// Конвейер шнековый 30330
	dks_shnek_30330:= x4_30;
	dp_shnek_30330:= NOT x4_31;
	localstop_shnek_30330:= NOT x5_0;
	erraz_shnek_30330:= NOT x5_1;
	localpusk_shnek_30330:= x5_2;
	y7_8:= run_shnek_30330;
	
// Затвор шлюзовый 30340
	dks_shluz_30340:= x5_3;
	erraz_shluz_30340:= NOT x5_4;
	y7_9:= run_shluz_30340;
	
// Конвейер скребковый 30400
	dks_sktr_30400:= x5_5;
	dp_sktr_30400:= NOT x5_6;
	localpusk_sktr_30400:= x5_7;
	localstop_sktr_30400:= NOT x5_8;
	localstop_end_sktr_30400:= NOT x5_9;
	erraz_sktr_30400:= NOT x5_10;
	y7_10:= run_sktr_30400;
	
// Нория 30500
	dks_noria_30500:= x5_11;
	dsl1_noria_30500:= NOT x5_12;
	dsl2_noria_30500:= NOT x5_13;
	dp_noria_30500:= NOT x5_14;
	localpusk_noria_30500:= x5_15;
	localstop_but_noria_30500:= NOT x5_16;
	localstop_top_noria_30500:= NOT x5_17;
	erraz_noria_30500:= NOT x5_18;
	y7_11:= run_noria_30500;	
	
// Датчики уровня бункеров смесителя
	TON_28(IN:= NOT x5_19, PT:= WORD_TO_TIME(timeDVY_load*100), Q=> dvy_bunk_30610);
	TON_29(IN:= NOT x5_20, PT:= WORD_TO_TIME(timeDNU_load*100), Q=> dny_bunk_30610);
	TON_30(IN:= NOT x5_21, PT:= WORD_TO_TIME(timeDNU_load*100), Q=> dny_bunk_30630);
	
// Датчик открытия люка на бункере БО-5	
	open_door_bunk_BO5:= x3_31;
	
// Смеситель горизонтальный СГП-1000 (30600)
	open_door_smes:= NOT x5_22;
	dks_smes:= x5_23;
	erraz_smes:= NOT x5_24;
	y7_12:= run_smes;
	
// от смесителя поворотный клапана, бомба люк
	klap_revers_open:= NOT x5_25;
	klap_revers_close:= NOT x5_26;
	shtok_1_left_open:= NOT x5_27;
	shtok_1_left_close:= NOT x5_28;
	shtok_2_left_open:= NOT x5_29;
	shtok_2_left_close:= NOT x5_30;
	shtok_1_right_open:= NOT x5_31;
	shtok_1_right_close:= NOT a2x0_0;
	shtok_2_right_open:= NOT a2x0_1;
	shtok_2_right_close:= NOT a2x0_2;
	shtok_1_zamok_close:= NOT a2x0_3;
	shtok_1_zamok_open:= NOT a2x0_4;
	shtok_2_zamok_close:= NOT a2x0_5;
	shtok_2_zamok_open:= NOT a2x0_6;
	signal_err_smes:= NOT a2x0_7;
	
	y7_13:= run_klap_revers_open;
	y7_14:= run_shtok_left_open;
	y7_15:= run_shtok_left_close;
	y7_16:= run_shtok_right_open;
	y7_17:= run_shtok_right_close;
	y7_18:= run_open_zamok;
	y7_19:= run_close_zamok;
	
// Конвейер шнековый 30640
	dks_shnek_30640:= a2x0_8;
	dp_shnek_30640:= NOT a2x0_9;
	localstop_shnek30640:= NOT a2x0_10;
	erraz_shnek_30640:= NOT a2x0_11;
	localpusk_shnek_30640:= a2x0_12;
	y7_20:= run_shnek_30640;
	
// Вентиляция аспирации АС7
	erraz_AC_7:= NOT a2x0_13;
	y7_21:= run_AC_7;
	
// Затвор шлюзовой аспирации АС-7_1
	dks_shluz_AC_7_1:= a2x0_14;
	erraz_shluz_AC_7_1:= NOT a2x0_15;
	y7_22:= run_shluz_AC_7_1;
	
// Затвор шлюзовой аспирации АС-7_2
	dks_shluz_AC_7_2:= a2x0_16;
	erraz_shluz_AC_7_2:= NOT a2x0_17;
	y7_23:= run_shluz_AC_7_2;
	
// Нория 30700
	dks_noria_30700:= a2x0_18;
	dsl1_noria_30700:= NOT a2x0_19;
	dsl2_noria_30700:= NOT a2x0_20;
	dp_noria_30700:= NOT a2x0_21;
	localpusk_noria_30700:= a2x0_22;
	localstop_but_noria_30700:= NOT a2x0_23;
	localstop_top_noria_30700:= NOT a2x3_0;
	erraz_noria_30700:= NOT a2x3_1;
	y7_24:= run_noria_30700;
	
// Система аспирации АС-8 (30701)
	erraz_AC_30701:= NOT a2x3_2;
	y7_25:= run_AC_30701;
	
// Конвейер скребковый 30900
	dp_sktr_30900:= NOT a2x3_3;
	localpusk_sktr_30900:= a2x3_4;
	localstop_sktr_30900:= NOT a2x3_5;
	erraz_sktr_30900:= NOT a2x3_6;
	dks_sktr_30900:= NOT a2x3_7;
	localstop_end_sktr_30900:= NOT a2x3_8;
	y7_26:= run_sktr_30900;
	
// Система аспирации АС-9 (30901)
	erraz_AC_30901:= NOT a2x3_9;
	y7_27:= run_AC_30901;
	
// Шибер конвейера 30900 (30910)
	opened_sh_30910:= NOT a2x3_10;
	closed_sh_30910:= NOT a2x3_11;
	erraz_sh_30910:= NOT a2x3_12;
	y7_28:= run_open_sh_30910;
	y7_29:= run_close_sh_30910;
	
// Шибер конвейера 30900 (30920)
	opened_sh_30920:= NOT a2x3_13;
	closed_sh_30920:= NOT a2x3_14;
	erraz_sh_30920:= NOT a2x3_15;
	y7_30:= run_open_sh_30920;
	y7_31:= run_close_sh_30920;
	
// Шибер конвейера 30900 (30930)
	opened_sh_30930:= NOT a2x3_16;
	closed_sh_30930:= NOT a2x3_17;
	erraz_sh_30930:= NOT a2x3_18;
	a2y0_0:= run_open_sh_30930;
	a2y0_1:= run_close_sh_30930;
	
// Шибер конвейера 30900 (30940)
	opened_sh_30940:= NOT a2x3_19;
	closed_sh_30940:= NOT a2x3_20;
	erraz_sh_30940:= NOT a2x3_21;
	a2y0_2:= run_open_sh_30940;
	a2y0_3:= run_close_sh_30940;
	
// Конвейер скребковыйй 30800
	dks_sktr_30800:= a2x3_22;
	dp_sktr_30800:= NOT a2x3_23;
	localpusk_sktr_30800:= a2x3_24;
	localstop_sktr_30800:= NOT a2x3_25;
	localstop_end_sktr_30800:= NOT a2x3_26;
	erraz_sktr_30800:= NOT a2x3_27;
	a2y0_4:= run_sktr_30800;
	
// Шибер конвейера 30800 (30810)
	opened_sh_30810:= NOT a2x3_28;
	closed_sh_30810:= NOT a2x3_29;
	erraz_sh_30810:= NOT a2x3_30;
	a2y0_5:= run_open_sh_30810;
	a2y0_6:= run_close_sh_30810;
	
// Конвейер бункера малых весов
	dks_shnek_21600:= a2x3_31;
	dp_shnek_21600:= NOT a2x4_0;
	localstop_21600:= NOT a2x4_1;
	erraz_shnek_21600:= NOT a2x4_2;
	localpusk_shnek_21600:= a2x4_3;
	a2y0_7:= run_shnek_21600;
	
// скальператор барабанный 10300
	errpch_scalp:= a2x4_4;
	a2y0_8:= run_scalp;
	a2y0_9:= run_resset_pch_scalp;
	a2y0_10:= run_pch_scalp;
	
// Дазаторы 20011-20016
	errpch_doz_11_16:= a2x4_5;
	a2y0_11:= run_pch_doz_11_16;
	a2y0_12:= run_resset_pch_doz_11_16;
	
	a2y0_13:= run_doz_shnek_20011;
	a2y0_14:= run_doz_shnek_20012;
	a2y0_15:= run_doz_shnek_20013;
	a2y6_0:= run_doz_shnek_20014;
	a2y6_1:= run_doz_shnek_20015;
	a2y6_2:= run_doz_shnek_20016;
	
	dp_doz_shnek_20011:= NOT a2x4_6;
	localstop_doz_shnek_20011:= NOT a2x4_7;
	dp_doz_shnek_20012:= NOT a2x4_8;
	localstop_doz_shnek_20012:= NOT a2x4_9;
	dp_doz_shnek_20013:= NOT a2x4_10;
	localstop_doz_shnek_20013:= NOT a2x4_11;
	dp_doz_shnek_20014:= NOT a2x4_12;
	localstop_doz_shnek_20014:= NOT a2x4_13;
	dp_doz_shnek_20015:= NOT a2x4_14;
	localstop_doz_shnek_20015:= NOT a2x4_15;
	dp_doz_shnek_20016:= NOT a2x4_16;
	localstop_doz_shnek_20016:= NOT a2x4_17;
	
// Дазаторы 20017-20018
	errpch_doz_17_18:= a2x4_18;
	a2y6_3:= run_pch_doz_17_18;
	a2y6_4:= run_resset_pch_doz_17_18;
	
	a2y6_5:= run_doz_shnek_20017;
	a2y6_6:= run_doz_shnek_20018;
	
	dp_doz_shnek_20017:= NOT a2x4_19;
	localstop_doz_shnek_20017:= NOT a2x4_20;
	dp_doz_shnek_20018:= NOT a2x4_21;
	localstop_doz_shnek_20018:= NOT a2x4_22;
	
// Дазатор 21510-21540
	errpch_doz_shnek_51_54:= a2x4_23;
	a2y6_7:= run_pch_doz_shnek_51_54;
	a2y6_8:= run_resset_pch_doz_shnek_51_54;
	
	a2y6_9:= run_doz_shnek_21510;
	a2y6_10:= run_doz_shnek_21520;
	a2y6_11:= run_doz_shnek_21530;
	a2y6_12:= run_doz_shnek_21540;
	
	dp_doz_shnek_21510:= NOT a2x4_24;
	localstop_doz_shnek_21510:= NOT a2x4_25;
	dp_doz_shnek_21520:= NOT a2x4_26;
	localstop_doz_shnek_21520:= NOT a2x4_27;
	dp_doz_shnek_21530:= NOT a2x4_28;
	localstop_doz_shnek_21530:= NOT a2x4_29;
	dp_doz_shnek_21540:= NOT a2x4_30;
	localstop_doz_shnek_21540:= NOT a2x4_31;
	
// Дазатор 21405-21409
	errpch_doz_shnek_5_9:= a2x5_0;
	a2y6_13:= run_pch_doz_shnek_5_9;
	a2y6_14:= run_resset_pch_doz_shnek_5_9;
	
	a2y6_15:= run_doz_shnek_21405;
	a2y6_16:= run_doz_shnek_21406;
	a2y6_17:= run_doz_shnek_21407;
	a2y6_18:= run_doz_shnek_21408;
	a2y6_19:= run_doz_shnek_21409;
	
	localstop_doz_shnek_21405:= NOT a2x5_1;
	localstop_doz_shnek_21406:= NOT a2x5_2;
	localstop_doz_shnek_21407:= NOT a2x5_3;
	localstop_doz_shnek_21408:= NOT a2x5_4;
	localstop_doz_shnek_21409:= NOT a2x5_5;
	
// Датчики верхнего уровня готовой продукции
	TON_31(IN:= NOT a2x5_6, PT:= WORD_TO_TIME(timeDVY_load*100), Q=> dvy_bunk_401);
	TON_32(IN:= NOT a2x5_7, PT:= WORD_TO_TIME(timeDVY_load*100), Q=> dvy_bunk_402);
	TON_33(IN:= NOT a2x5_8, PT:= WORD_TO_TIME(timeDVY_load*100), Q=> dvy_bunk_403);
	TON_34(IN:= NOT a2x5_9, PT:= WORD_TO_TIME(timeDVY_load*100), Q=> dvy_bunk_404);
	TON_35(IN:= NOT a2x5_10, PT:= WORD_TO_TIME(timeDVY_load*100), Q=> dvy_bunk_405);
	TON_36(IN:= NOT a2x5_11, PT:= WORD_TO_TIME(timeDVY_load*100), Q=> dvy_bunk_406);

// Датчики нижнего уровня готовой продукции
	TON_37(IN:= NOT a2x5_12, PT:= WORD_TO_TIME(timeDNU_load*100), Q=> dny_bunk_401);
	TON_38(IN:= NOT a2x5_13, PT:= WORD_TO_TIME(timeDNU_load*100), Q=> dny_bunk_402);
	TON_39(IN:= NOT a2x5_14, PT:= WORD_TO_TIME(timeDNU_load*100), Q=> dny_bunk_403);
	TON_40(IN:= NOT a2x5_15, PT:= WORD_TO_TIME(timeDNU_load*100), Q=> dny_bunk_404);
	TON_41(IN:= NOT a2x5_16, PT:= WORD_TO_TIME(timeDNU_load*100), Q=> dny_bunk_405);
	TON_42(IN:= NOT a2x5_17, PT:= WORD_TO_TIME(timeDNU_load*100), Q=> dny_bunk_406);
	
// Вентиляторы фильтр-шкафоф завальной ямы
	localpusk_fan_hole:= a2x5_18;
	localstop_fan_hole:= NOT a2x5_19;
	erraz_AC1_1_1:= NOT a2x5_20;
	erraz_AC2_1_1:= NOT a2x5_21;
	erraz_AC3_1_1:= NOT a2x5_22;
	erraz_AC1_1_2:= NOT a2x5_23;
	erraz_AC2_1_2:= NOT a2x5_24;
	erraz_AC3_1_2:= NOT a2x5_25;
	a2y6_20:= run_fans_AC_hole;
	
// Датчик нижнего уровня завальной ямы
	TON_43(IN:= NOT a2x5_26, PT:= WORD_TO_TIME(timeDNU_load*100), Q=> dny_hole);
	
// Конвейер 30330
	errpch_sktr_30330:= a2x5_27;
	a2y6_21:= run_pch_sktr_30330;
	a2y6_22:= run_resset_pch_sktr_30330;
	
// Конвейер 30640
	errpch_sktr_30640:= a2x5_28;
	a2y6_23:= run_pch_sktr_30640;
	a2y6_24:= run_resset_pch_sktr_30640;
	
// Весы большие
	W1_Big:= %IW39;
	W2_Big:= %IW40;
	Weight_Big.WordValue[0]:= W2_Big;
	Weight_Big.WordValue[1]:= W1_Big;
	CurrWeight_Big:= Weight_Big.RealValue-Tare_big_weight;
	
// Весы средние
	W1_Midle:= %IW41;
	W2_Midle:= %IW42;
	Weight_Midle.WordValue[0]:= W2_Midle;
	Weight_Midle.WordValue[1]:= W1_Midle;
	CurrWeight_Midle:= Weight_Midle.RealValue-Tare_midle_weight;

END_PROGRAM

// PLC_241/Application/POU/prgLoad
PROGRAM prgLoad
VAR
	T_SKTR_10110: T;
	AC_10201: AC;
	N_10200: N;
	KP_10210: KP;
	SCLP_10300: SCLP;
	AC_10401: AC;
	N_10400: N;
	AC_10501: AC;
	T_10500: T;
	Z_10610: Z;
	KP_10710: KP;
	Z_10620: Z;
	KP_10720: KP;
	Z_10630: Z;
	KP_10730: KP;
	Z_10640: Z;
	KP_10740: KP;
	AC_fans_hole: AC;
	TP_STEP: TP;
	Step: WORD;
	imp: BOOL;
	imp_dvy_101: BOOL;
	imp_dvy_102: BOOL;
	imp_dvy_103: BOOL;
	imp_dvy_104: BOOL;
	imp_dvy_105: BOOL;
	imp_dvy_106: BOOL;
	imp_dvy_107: BOOL;
	imp_dvy_108: BOOL;
	pause_load: BOOL;
	TON_pause: TON;
	TOF_next_sktr_10500: TOF;
	TON_imp_bunk_101: TON;
	TON_imp_bunk_102: TON;
	timePause_load_queu3: TON;
	TON_imp_bunk_103: TON;
	TON_imp_bunk_104: TON;
	TON_imp_bunk_105: TON;
	TON_imp_bunk_107: TON;
	TON_imp_bunk_106: TON;
	TON_imp_bunk_108: TON;
	TON_pause_DNY_HOLE: TON;
	use_time_hole: BOOL;
	TON_RESSET_modeLoad: TON;
	check: BOOL;
	TON_nextBunk: TON;
	imp_nextBunk: BOOL;
END_VAR
VAR // added by the converter: edge detectors and wires of the graphical bodies
    _rt1, _rt2, _rt3, _rt4, _rt5, _rt6, _rt7, _rt8, _rt9, _rt10, _rt11, _rt12, _rt13, _rt14, _rt15, _rt16, _rt17, _rt18, _rt19, _rt20, _rt21 : R_TRIG;
    _w1, _w2, _w3, _w4, _w5, _w6, _w7, _w8, _w9, _w10 : BOOL;
END_VAR

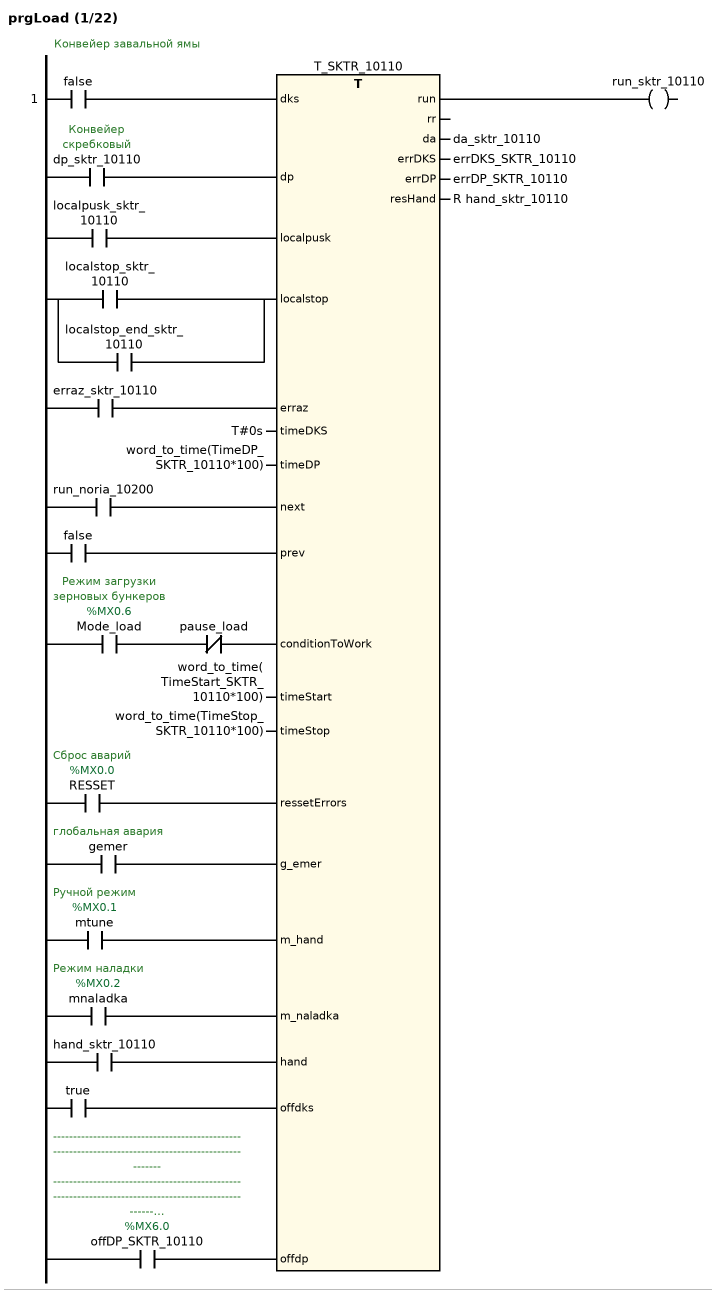
// NETWORK 1
// Конвейер завальной ямы
//   dp_sktr_10110: Конвейер скребковый
//   Mode_load: Режим загрузки зерновых бункеров | AT %MX0.6
//   RESSET: Сброс аварий | AT %MX0.0
//   gemer: глобальная авария
//   mtune: Ручной режим | AT %MX0.1
//   mnaladka: Режим наладки | AT %MX0.2
//   offDP_SKTR_10110: ----------------------------------------------------------------------------------------------------- ----------------------------------------------------------------------------------------------------- Отключение датчиков из скады ----------------------------------------------------------------------------------------------------- Конвейер завальной ямы | AT %MX6.0
//   errDKS_SKTR_10110: Конвейер завальной ямы 10110
T_SKTR_10110(
    dks := false,
    dp := dp_sktr_10110,
    localpusk := localpusk_sktr_10110,
    localstop := localstop_sktr_10110 OR localstop_end_sktr_10110,
    erraz := erraz_sktr_10110,
    timeDKS := T#0s,
    timeDP := word_to_time(TimeDP_SKTR_10110*100),
    next := run_noria_10200,
    prev := false,
    conditionToWork := Mode_load AND NOT pause_load,
    timeStart := word_to_time(TimeStart_SKTR_10110*100),
    timeStop := word_to_time(TimeStop_SKTR_10110*100),
    ressetErrors := RESSET,
    g_emer := gemer,
    m_hand := mtune,
    m_naladka := mnaladka,
    hand := hand_sktr_10110,
    offdks := true,
    offdp := offDP_SKTR_10110,
    da => da_sktr_10110,
    errDKS => errDKS_SKTR_10110,
    errDP => errDP_SKTR_10110); // T
hand_sktr_10110 R= T_SKTR_10110.resHand;
run_sktr_10110 := T_SKTR_10110.run;

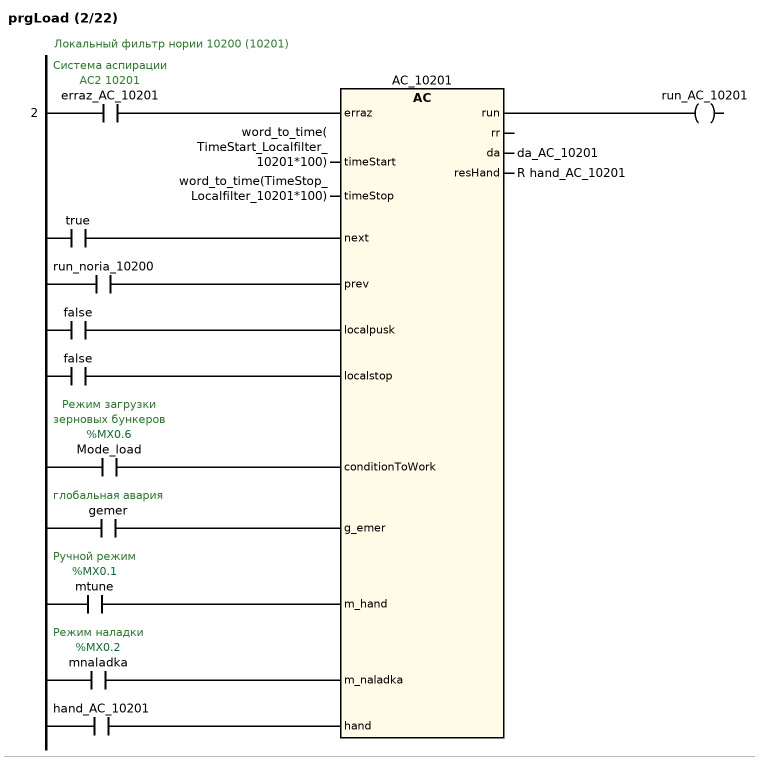
// NETWORK 2
// Локальный фильтр нории 10200 (10201)
//   erraz_AC_10201: Система аспирации АС2 10201
//   Mode_load: Режим загрузки зерновых бункеров | AT %MX0.6
//   gemer: глобальная авария
//   mtune: Ручной режим | AT %MX0.1
//   mnaladka: Режим наладки | AT %MX0.2
AC_10201(
    erraz := erraz_AC_10201,
    timeStart := word_to_time(TimeStart_Localfilter_10201*100),
    timeStop := word_to_time(TimeStop_Localfilter_10201*100),
    next := true,
    prev := run_noria_10200,
    localpusk := false,
    localstop := false,
    conditionToWork := Mode_load,
    g_emer := gemer,
    m_hand := mtune,
    m_naladka := mnaladka,
    hand := hand_AC_10201,
    da => da_AC_10201); // AC
hand_AC_10201 R= AC_10201.resHand;
run_AC_10201 := AC_10201.run;

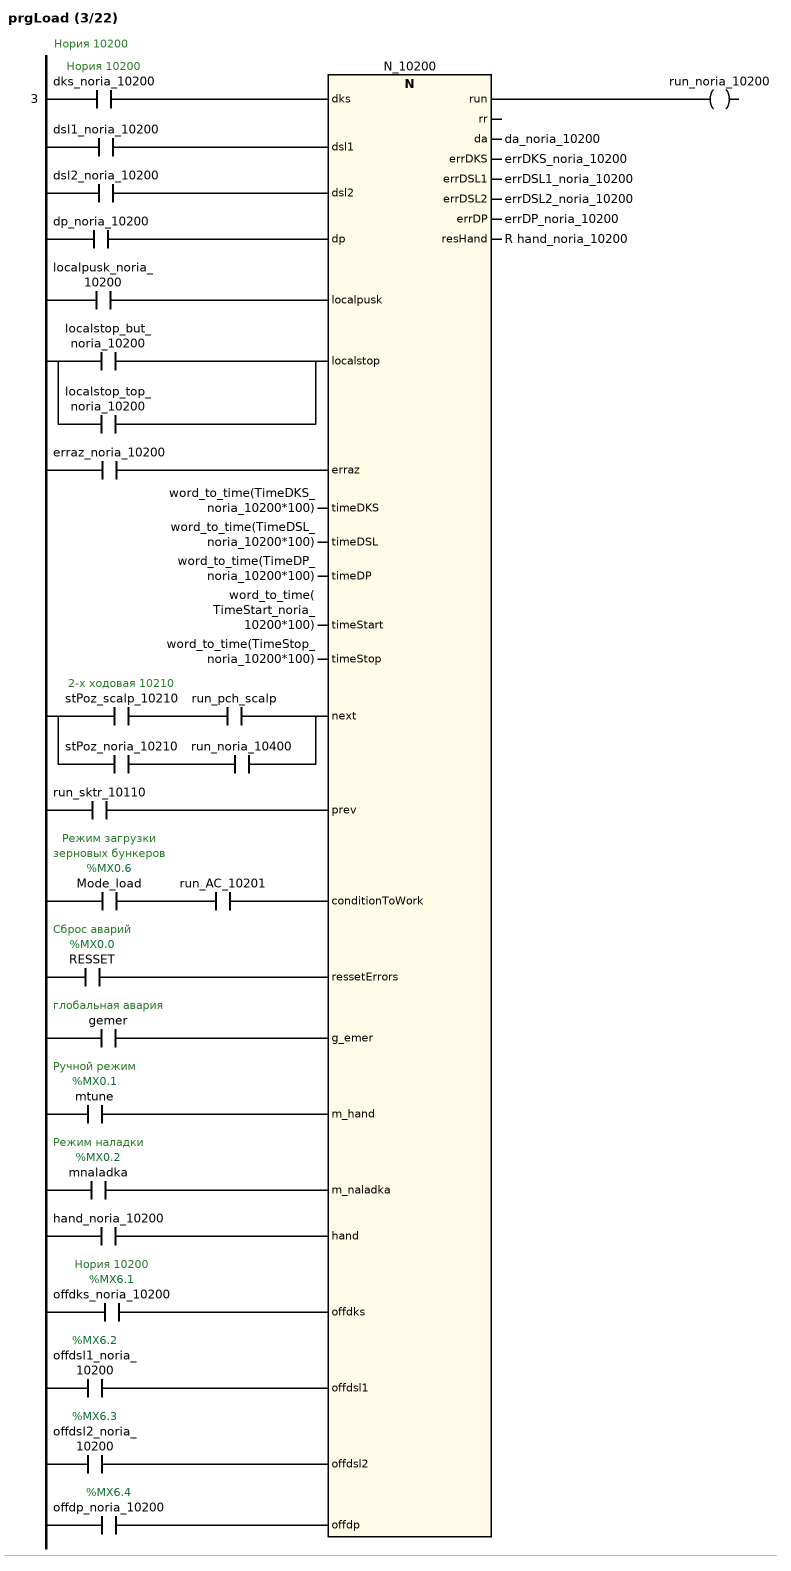
// NETWORK 3
// Нория 10200
//   dks_noria_10200: Нория 10200
//   stPoz_scalp_10210: 2-х ходовая 10210
//   Mode_load: Режим загрузки зерновых бункеров | AT %MX0.6
//   RESSET: Сброс аварий | AT %MX0.0
//   gemer: глобальная авария
//   mtune: Ручной режим | AT %MX0.1
//   mnaladka: Режим наладки | AT %MX0.2
//   offdks_noria_10200: Нория 10200 | AT %MX6.1
//   offdsl1_noria_10200: AT %MX6.2
//   offdsl2_noria_10200: AT %MX6.3
//   offdp_noria_10200: AT %MX6.4
//   errDKS_noria_10200: Нория 10200
N_10200(
    dks := dks_noria_10200,
    dsl1 := dsl1_noria_10200,
    dsl2 := dsl2_noria_10200,
    dp := dp_noria_10200,
    localpusk := localpusk_noria_10200,
    localstop := localstop_but_noria_10200 OR localstop_top_noria_10200,
    erraz := erraz_noria_10200,
    timeDKS := word_to_time(TimeDKS_noria_10200*100),
    timeDSL := word_to_time(TimeDSL_noria_10200*100),
    timeDP := word_to_time(TimeDP_noria_10200*100),
    timeStart := word_to_time(TimeStart_noria_10200*100),
    timeStop := word_to_time(TimeStop_noria_10200*100),
    next := stPoz_scalp_10210 AND run_pch_scalp OR stPoz_noria_10210 AND run_noria_10400,
    prev := run_sktr_10110,
    conditionToWork := Mode_load AND run_AC_10201,
    ressetErrors := RESSET,
    g_emer := gemer,
    m_hand := mtune,
    m_naladka := mnaladka,
    hand := hand_noria_10200,
    offdks := offdks_noria_10200,
    offdsl1 := offdsl1_noria_10200,
    offdsl2 := offdsl2_noria_10200,
    offdp := offdp_noria_10200,
    da => da_noria_10200,
    errDKS => errDKS_noria_10200,
    errDSL1 => errDSL1_noria_10200,
    errDSL2 => errDSL2_noria_10200,
    errDP => errDP_noria_10200); // N
hand_noria_10200 R= N_10200.resHand;
run_noria_10200 := N_10200.run;

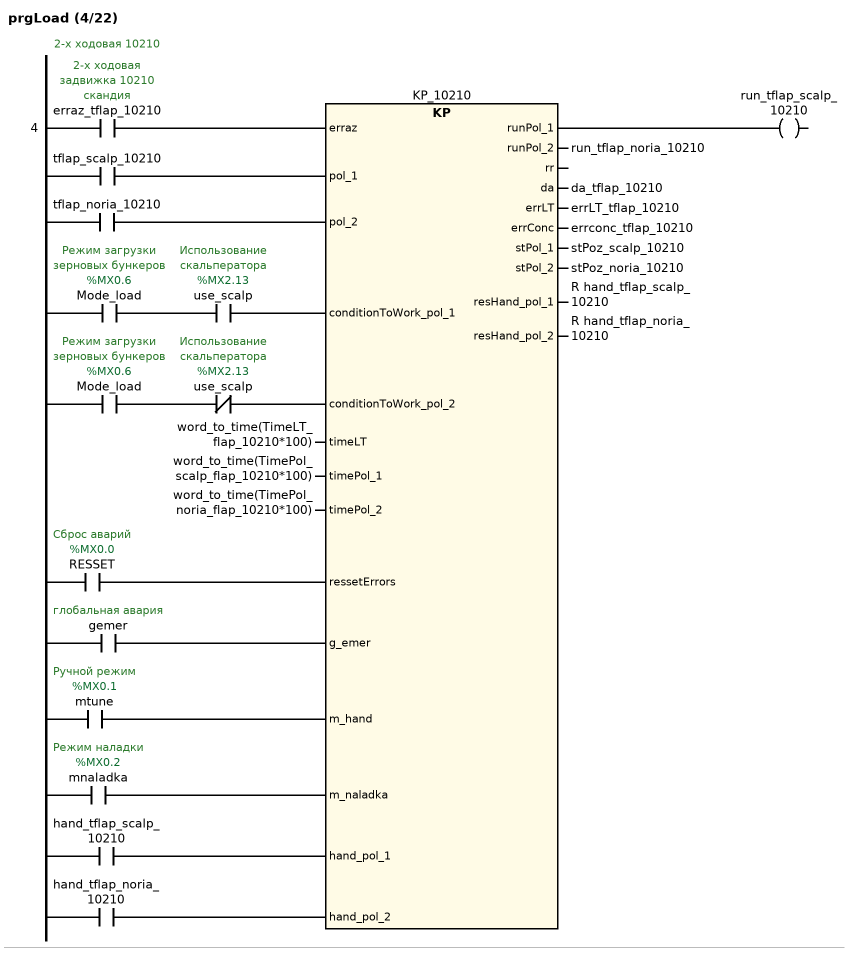
// NETWORK 4
// 2-х ходовая 10210
//   erraz_tflap_10210: 2-х ходовая задвижка 10210 скандия
//   Mode_load: Режим загрузки зерновых бункеров | AT %MX0.6
//   use_scalp: Использование скальператора | AT %MX2.13
//   RESSET: Сброс аварий | AT %MX0.0
//   gemer: глобальная авария
//   mtune: Ручной режим | AT %MX0.1
//   mnaladka: Режим наладки | AT %MX0.2
//   errLT_tflap_10210: 2-х ходовой клапан КП_10210
//   stPoz_scalp_10210: 2-х ходовая 10210
KP_10210(
    erraz := erraz_tflap_10210,
    pol_1 := tflap_scalp_10210,
    pol_2 := tflap_noria_10210,
    conditionToWork_pol_1 := Mode_load AND use_scalp,
    conditionToWork_pol_2 := Mode_load AND NOT use_scalp,
    timeLT := word_to_time(TimeLT_flap_10210*100),
    timePol_1 := word_to_time(TimePol_scalp_flap_10210*100),
    timePol_2 := word_to_time(TimePol_noria_flap_10210*100),
    ressetErrors := RESSET,
    g_emer := gemer,
    m_hand := mtune,
    m_naladka := mnaladka,
    hand_pol_1 := hand_tflap_scalp_10210,
    hand_pol_2 := hand_tflap_noria_10210,
    runPol_2 => run_tflap_noria_10210,
    da => da_tflap_10210,
    errLT => errLT_tflap_10210,
    errConc => errconc_tflap_10210,
    stPol_1 => stPoz_scalp_10210,
    stPol_2 => stPoz_noria_10210); // KP
hand_tflap_scalp_10210 R= KP_10210.resHand_pol_1;
hand_tflap_noria_10210 R= KP_10210.resHand_pol_2;
run_tflap_scalp_10210 := KP_10210.runPol_1;

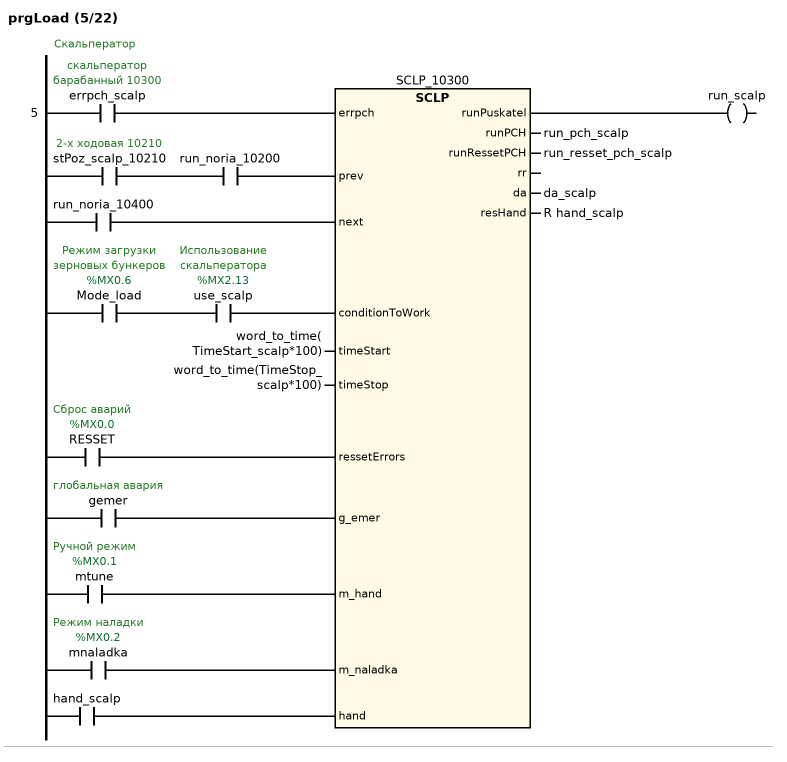
// NETWORK 5
// Скальператор
//   errpch_scalp: скальператор барабанный 10300
//   stPoz_scalp_10210: 2-х ходовая 10210
//   Mode_load: Режим загрузки зерновых бункеров | AT %MX0.6
//   use_scalp: Использование скальператора | AT %MX2.13
//   RESSET: Сброс аварий | AT %MX0.0
//   gemer: глобальная авария
//   mtune: Ручной режим | AT %MX0.1
//   mnaladka: Режим наладки | AT %MX0.2
SCLP_10300(
    errpch := errpch_scalp,
    prev := stPoz_scalp_10210 AND run_noria_10200,
    next := run_noria_10400,
    conditionToWork := Mode_load AND use_scalp,
    timeStart := word_to_time(TimeStart_scalp*100),
    timeStop := word_to_time(TimeStop_scalp*100),
    ressetErrors := RESSET,
    g_emer := gemer,
    m_hand := mtune,
    m_naladka := mnaladka,
    hand := hand_scalp,
    runPCH => run_pch_scalp,
    runRessetPCH => run_resset_pch_scalp,
    da => da_scalp); // SCLP
hand_scalp R= SCLP_10300.resHand;
run_scalp := SCLP_10300.runPuskatel;

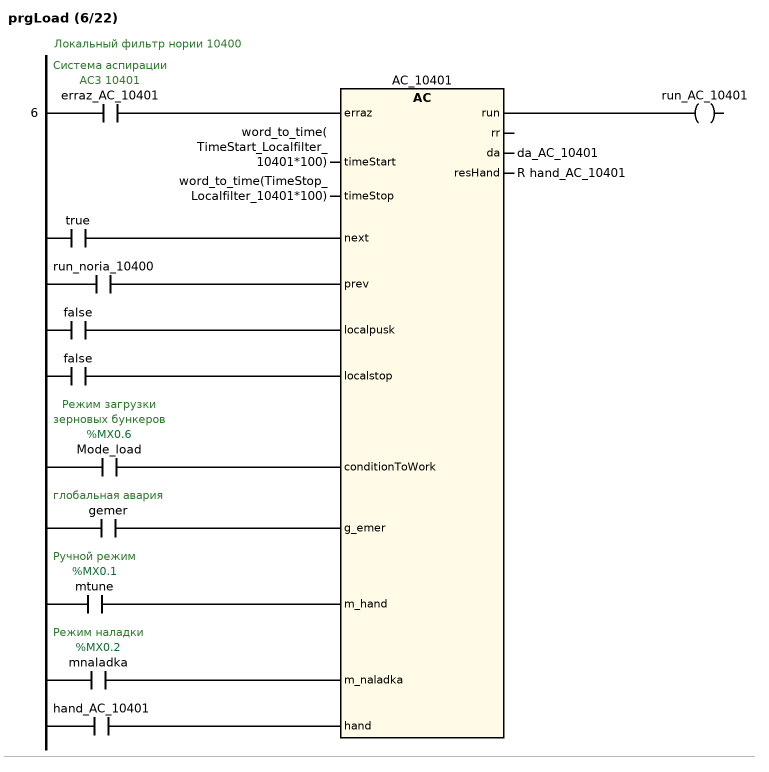
// NETWORK 6
// Локальный фильтр нории 10400
//   erraz_AC_10401: Система аспирации АС3 10401
//   Mode_load: Режим загрузки зерновых бункеров | AT %MX0.6
//   gemer: глобальная авария
//   mtune: Ручной режим | AT %MX0.1
//   mnaladka: Режим наладки | AT %MX0.2
AC_10401(
    erraz := erraz_AC_10401,
    timeStart := word_to_time(TimeStart_Localfilter_10401*100),
    timeStop := word_to_time(TimeStop_Localfilter_10401*100),
    next := true,
    prev := run_noria_10400,
    localpusk := false,
    localstop := false,
    conditionToWork := Mode_load,
    g_emer := gemer,
    m_hand := mtune,
    m_naladka := mnaladka,
    hand := hand_AC_10401,
    da => da_AC_10401); // AC
hand_AC_10401 R= AC_10401.resHand;
run_AC_10401 := AC_10401.run;

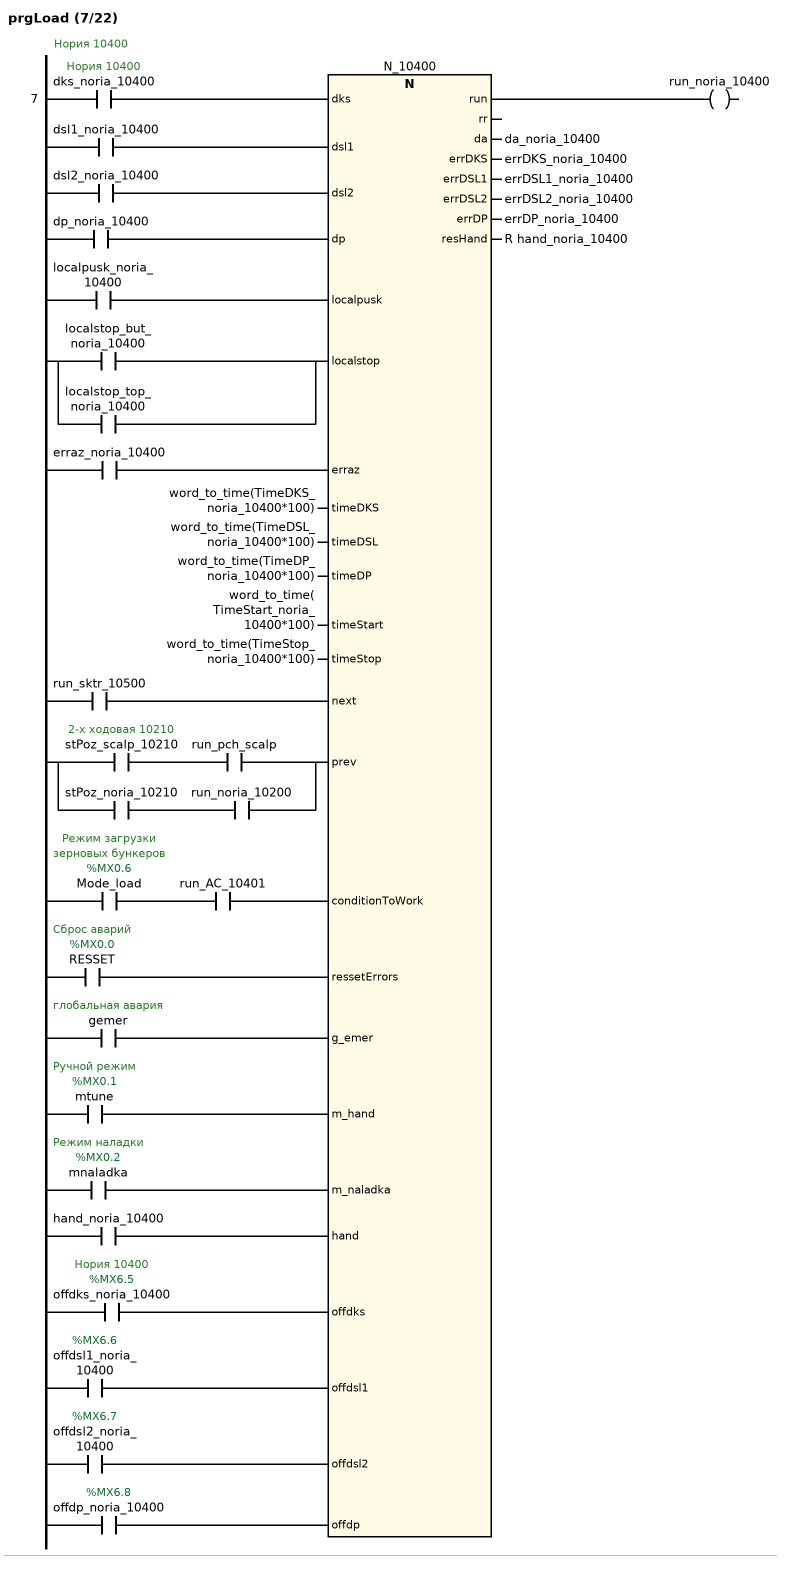
// NETWORK 7
// Нория 10400
//   dks_noria_10400: Нория 10400
//   stPoz_scalp_10210: 2-х ходовая 10210
//   Mode_load: Режим загрузки зерновых бункеров | AT %MX0.6
//   RESSET: Сброс аварий | AT %MX0.0
//   gemer: глобальная авария
//   mtune: Ручной режим | AT %MX0.1
//   mnaladka: Режим наладки | AT %MX0.2
//   offdks_noria_10400: Нория 10400 | AT %MX6.5
//   offdsl1_noria_10400: AT %MX6.6
//   offdsl2_noria_10400: AT %MX6.7
//   offdp_noria_10400: AT %MX6.8
//   errDKS_noria_10400: Нория 10400
N_10400(
    dks := dks_noria_10400,
    dsl1 := dsl1_noria_10400,
    dsl2 := dsl2_noria_10400,
    dp := dp_noria_10400,
    localpusk := localpusk_noria_10400,
    localstop := localstop_but_noria_10400 OR localstop_top_noria_10400,
    erraz := erraz_noria_10400,
    timeDKS := word_to_time(TimeDKS_noria_10400*100),
    timeDSL := word_to_time(TimeDSL_noria_10400*100),
    timeDP := word_to_time(TimeDP_noria_10400*100),
    timeStart := word_to_time(TimeStart_noria_10400*100),
    timeStop := word_to_time(TimeStop_noria_10400*100),
    next := run_sktr_10500,
    prev := stPoz_scalp_10210 AND run_pch_scalp OR stPoz_noria_10210 AND run_noria_10200,
    conditionToWork := Mode_load AND run_AC_10401,
    ressetErrors := RESSET,
    g_emer := gemer,
    m_hand := mtune,
    m_naladka := mnaladka,
    hand := hand_noria_10400,
    offdks := offdks_noria_10400,
    offdsl1 := offdsl1_noria_10400,
    offdsl2 := offdsl2_noria_10400,
    offdp := offdp_noria_10400,
    da => da_noria_10400,
    errDKS => errDKS_noria_10400,
    errDSL1 => errDSL1_noria_10400,
    errDSL2 => errDSL2_noria_10400,
    errDP => errDP_noria_10400); // N
hand_noria_10400 R= N_10400.resHand;
run_noria_10400 := N_10400.run;

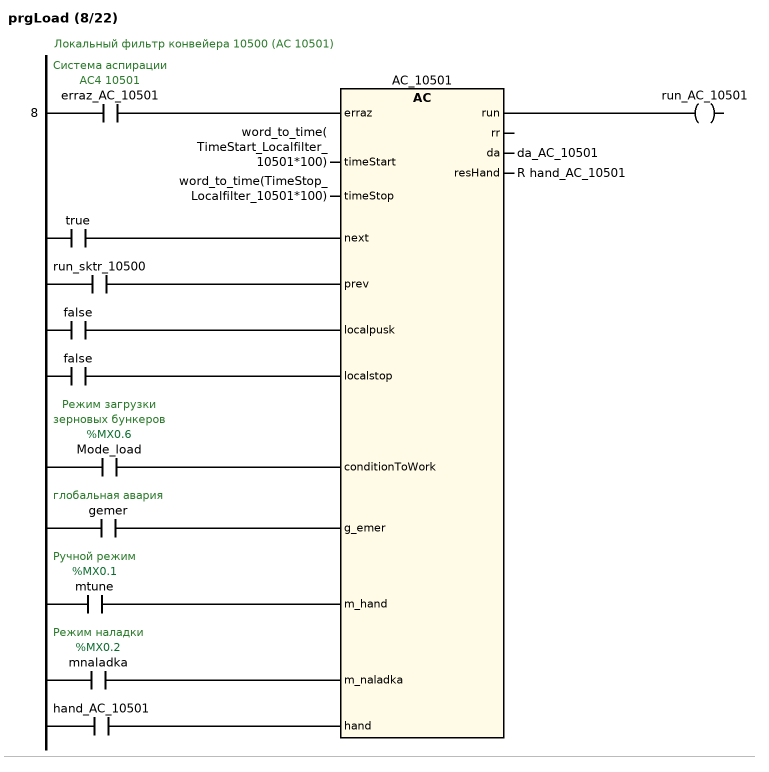
// NETWORK 8
// Локальный фильтр конвейера 10500 (АС 10501)
//   erraz_AC_10501: Система аспирации АС4 10501
//   Mode_load: Режим загрузки зерновых бункеров | AT %MX0.6
//   gemer: глобальная авария
//   mtune: Ручной режим | AT %MX0.1
//   mnaladka: Режим наладки | AT %MX0.2
AC_10501(
    erraz := erraz_AC_10501,
    timeStart := word_to_time(TimeStart_Localfilter_10501*100),
    timeStop := word_to_time(TimeStop_Localfilter_10501*100),
    next := true,
    prev := run_sktr_10500,
    localpusk := false,
    localstop := false,
    conditionToWork := Mode_load,
    g_emer := gemer,
    m_hand := mtune,
    m_naladka := mnaladka,
    hand := hand_AC_10501,
    da => da_AC_10501); // AC
hand_AC_10501 R= AC_10501.resHand;
run_AC_10501 := AC_10501.run;

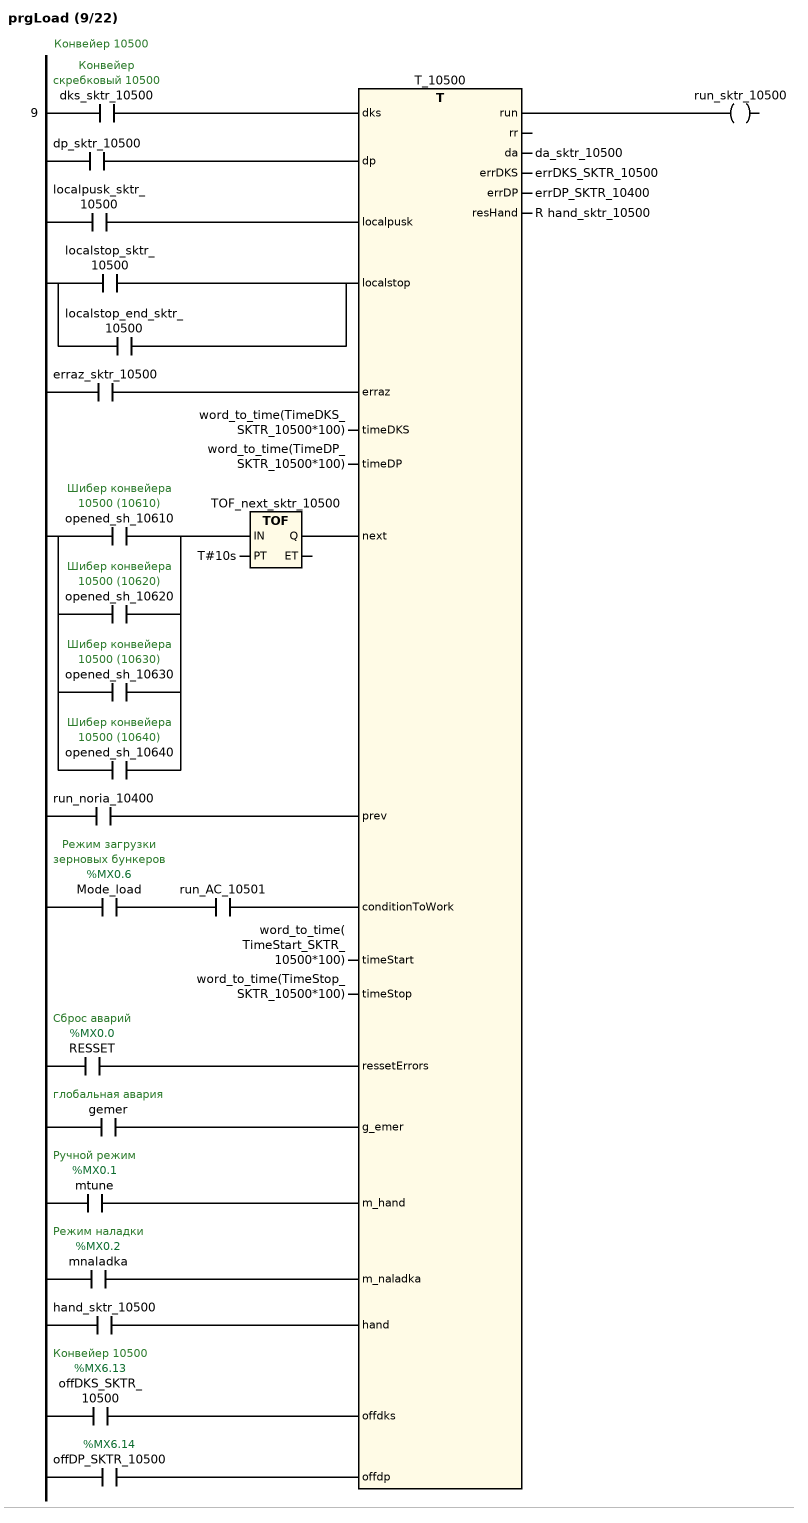
// NETWORK 9
// Конвейер 10500
//   dks_sktr_10500: Конвейер скребковый 10500
//   opened_sh_10610: Шибер конвейера 10500 (10610)
//   opened_sh_10620: Шибер конвейера 10500 (10620)
//   opened_sh_10630: Шибер конвейера 10500 (10630)
//   opened_sh_10640: Шибер конвейера 10500 (10640)
//   Mode_load: Режим загрузки зерновых бункеров | AT %MX0.6
//   RESSET: Сброс аварий | AT %MX0.0
//   gemer: глобальная авария
//   mtune: Ручной режим | AT %MX0.1
//   mnaladka: Режим наладки | AT %MX0.2
//   offDKS_SKTR_10500: Конвейер 10500 | AT %MX6.13
//   offDP_SKTR_10500: AT %MX6.14
//   errDKS_SKTR_10500: Конвейер 10500
TOF_next_sktr_10500(IN := opened_sh_10610 OR opened_sh_10620 OR opened_sh_10630 OR opened_sh_10640, PT := T#10s); // TOF
T_10500(
    dks := dks_sktr_10500,
    dp := dp_sktr_10500,
    localpusk := localpusk_sktr_10500,
    localstop := localstop_sktr_10500 OR localstop_end_sktr_10500,
    erraz := erraz_sktr_10500,
    timeDKS := word_to_time(TimeDKS_SKTR_10500*100),
    timeDP := word_to_time(TimeDP_SKTR_10500*100),
    next := TOF_next_sktr_10500.Q,
    prev := run_noria_10400,
    conditionToWork := Mode_load AND run_AC_10501,
    timeStart := word_to_time(TimeStart_SKTR_10500*100),
    timeStop := word_to_time(TimeStop_SKTR_10500*100),
    ressetErrors := RESSET,
    g_emer := gemer,
    m_hand := mtune,
    m_naladka := mnaladka,
    hand := hand_sktr_10500,
    offdks := offDKS_SKTR_10500,
    offdp := offDP_SKTR_10500,
    da => da_sktr_10500,
    errDKS => errDKS_SKTR_10500,
    errDP => errDP_SKTR_10400); // T
hand_sktr_10500 R= T_10500.resHand;
run_sktr_10500 := T_10500.run;

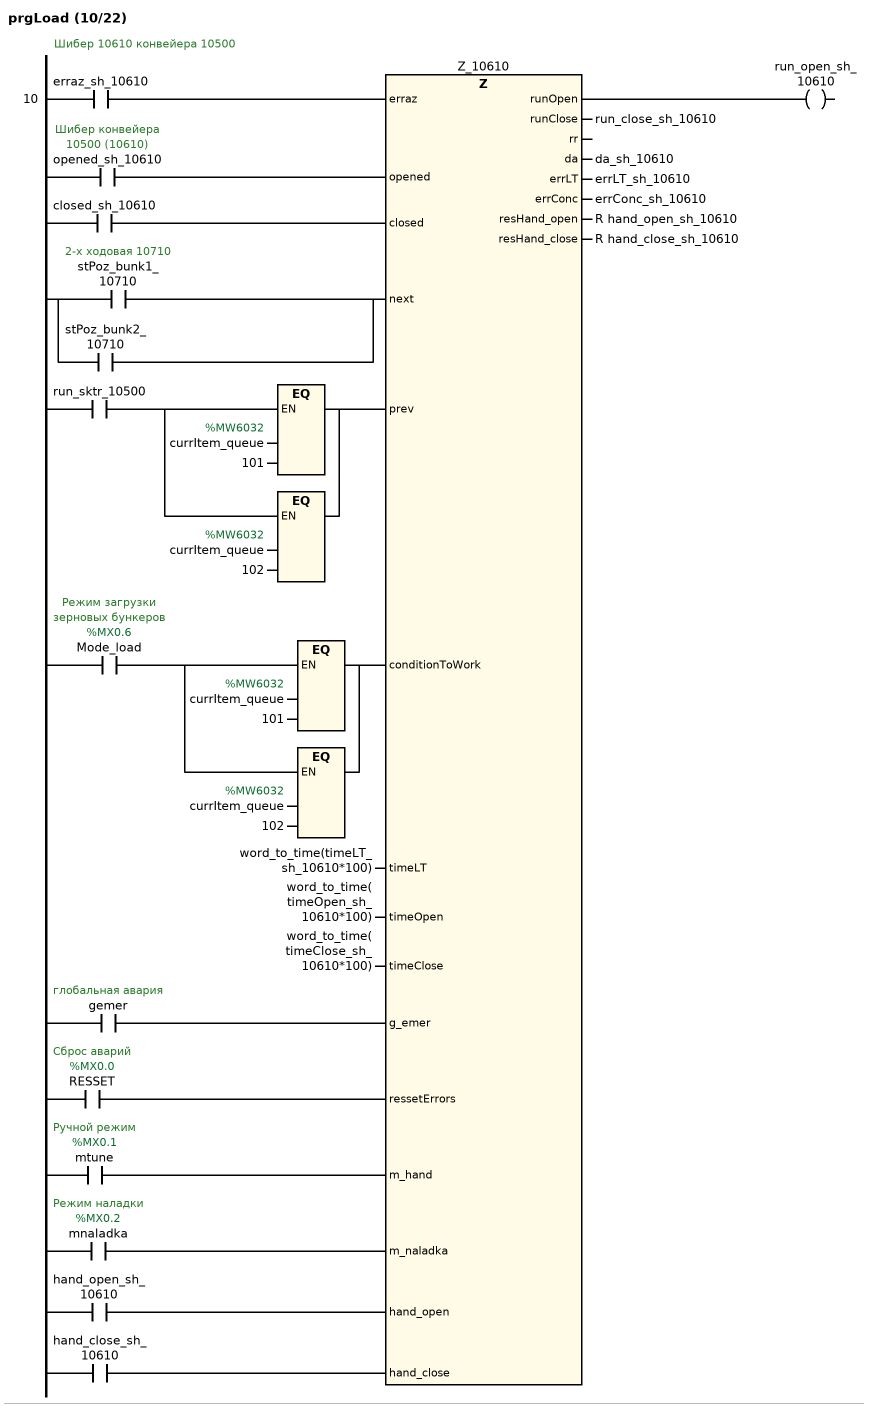
// NETWORK 10
// Шибер 10610 конвейера 10500
//   opened_sh_10610: Шибер конвейера 10500 (10610)
//   stPoz_bunk1_10710: 2-х ходовая 10710
//   currItem_queue: Текущий бункер для загрузки в очереди | AT %MW6032
//   Mode_load: Режим загрузки зерновых бункеров | AT %MX0.6
//   gemer: глобальная авария
//   RESSET: Сброс аварий | AT %MX0.0
//   mtune: Ручной режим | AT %MX0.1
//   mnaladka: Режим наладки | AT %MX0.2
//   errLT_sh_10610: Шибер 10610
Z_10610(
    erraz := erraz_sh_10610,
    opened := opened_sh_10610,
    closed := closed_sh_10610,
    next := stPoz_bunk1_10710 OR stPoz_bunk2_10710,
    prev := run_sktr_10500 AND currItem_queue = 101 OR run_sktr_10500 AND currItem_queue = 102,
    conditionToWork := Mode_load AND currItem_queue = 101 OR Mode_load AND currItem_queue = 102,
    timeLT := word_to_time(timeLT_sh_10610*100),
    timeOpen := word_to_time(timeOpen_sh_10610*100),
    timeClose := word_to_time(timeClose_sh_10610*100),
    g_emer := gemer,
    ressetErrors := RESSET,
    m_hand := mtune,
    m_naladka := mnaladka,
    hand_open := hand_open_sh_10610,
    hand_close := hand_close_sh_10610,
    runClose => run_close_sh_10610,
    da => da_sh_10610,
    errLT => errLT_sh_10610,
    errConc => errConc_sh_10610); // Z
hand_open_sh_10610 R= Z_10610.resHand_open;
hand_close_sh_10610 R= Z_10610.resHand_close;
run_open_sh_10610 := Z_10610.runOpen;

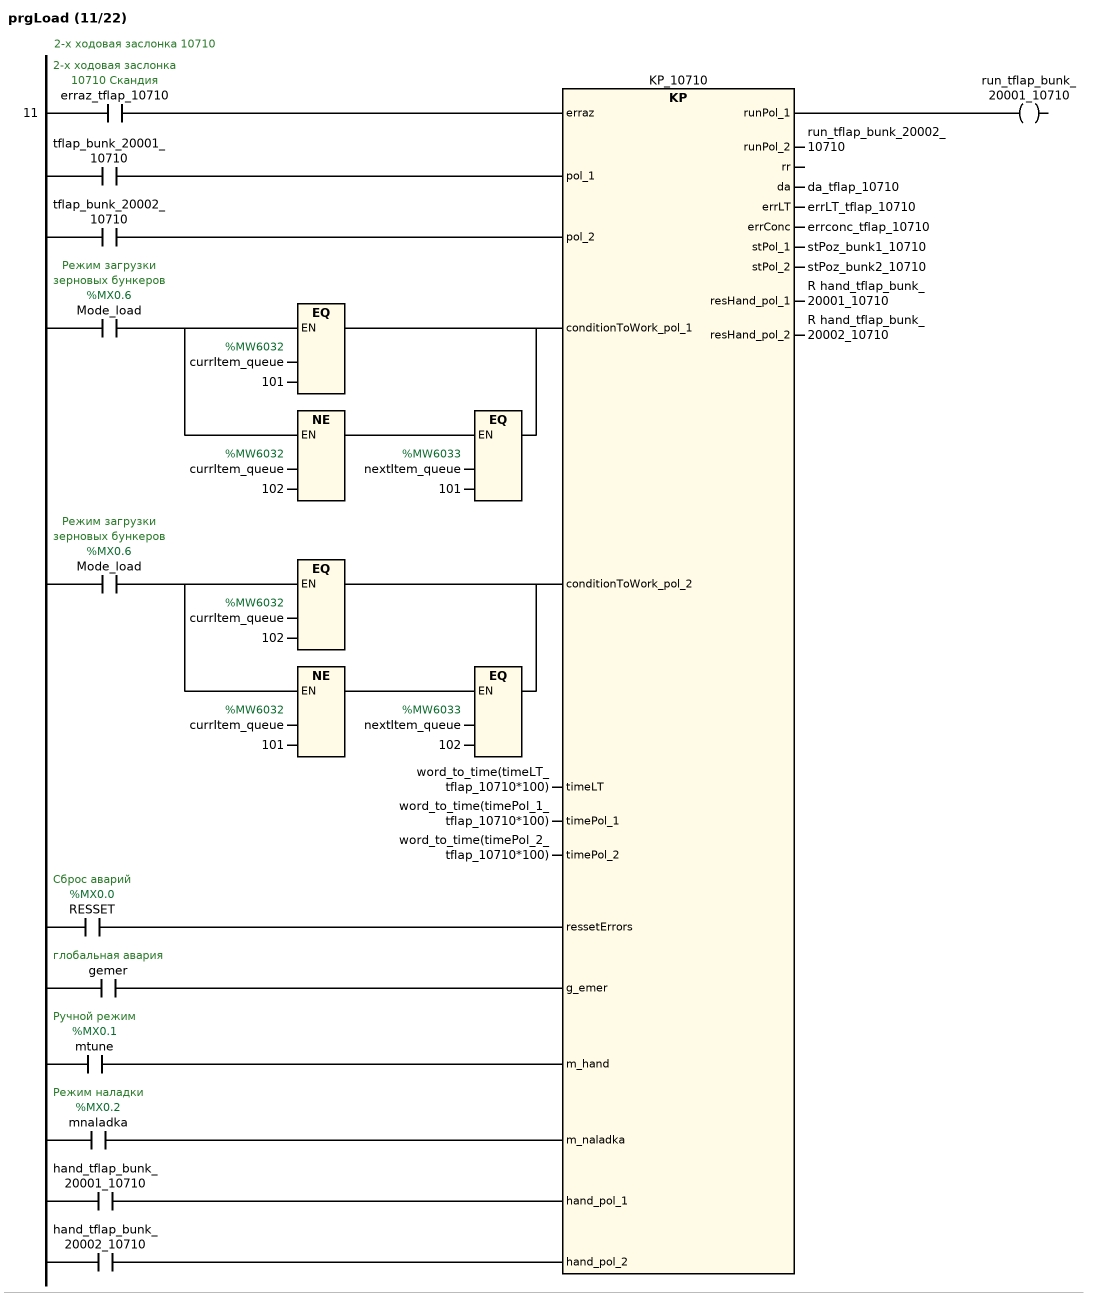
// NETWORK 11
// 2-х ходовая заслонка 10710
//   erraz_tflap_10710: 2-х ходовая заслонка 10710 Скандия
//   Mode_load: Режим загрузки зерновых бункеров | AT %MX0.6
//   currItem_queue: Текущий бункер для загрузки в очереди | AT %MW6032
//   nextItem_queue: Следующий бункер для загрузки в очереди | AT %MW6033
//   RESSET: Сброс аварий | AT %MX0.0
//   gemer: глобальная авария
//   mtune: Ручной режим | AT %MX0.1
//   mnaladka: Режим наладки | AT %MX0.2
//   errLT_tflap_10710: 2-х ходовой клапан КП_10710
//   stPoz_bunk1_10710: 2-х ходовая 10710
KP_10710(
    erraz := erraz_tflap_10710,
    pol_1 := tflap_bunk_20001_10710,
    pol_2 := tflap_bunk_20002_10710,
    conditionToWork_pol_1 := Mode_load AND currItem_queue = 101 OR Mode_load AND currItem_queue <> 102 AND nextItem_queue = 101,
    conditionToWork_pol_2 := Mode_load AND currItem_queue = 102 OR Mode_load AND currItem_queue <> 101 AND nextItem_queue = 102,
    timeLT := word_to_time(timeLT_tflap_10710*100),
    timePol_1 := word_to_time(timePol_1_tflap_10710*100),
    timePol_2 := word_to_time(timePol_2_tflap_10710*100),
    ressetErrors := RESSET,
    g_emer := gemer,
    m_hand := mtune,
    m_naladka := mnaladka,
    hand_pol_1 := hand_tflap_bunk_20001_10710,
    hand_pol_2 := hand_tflap_bunk_20002_10710,
    runPol_2 => run_tflap_bunk_20002_10710,
    da => da_tflap_10710,
    errLT => errLT_tflap_10710,
    errConc => errconc_tflap_10710,
    stPol_1 => stPoz_bunk1_10710,
    stPol_2 => stPoz_bunk2_10710); // KP
hand_tflap_bunk_20001_10710 R= KP_10710.resHand_pol_1;
hand_tflap_bunk_20002_10710 R= KP_10710.resHand_pol_2;
run_tflap_bunk_20001_10710 := KP_10710.runPol_1;

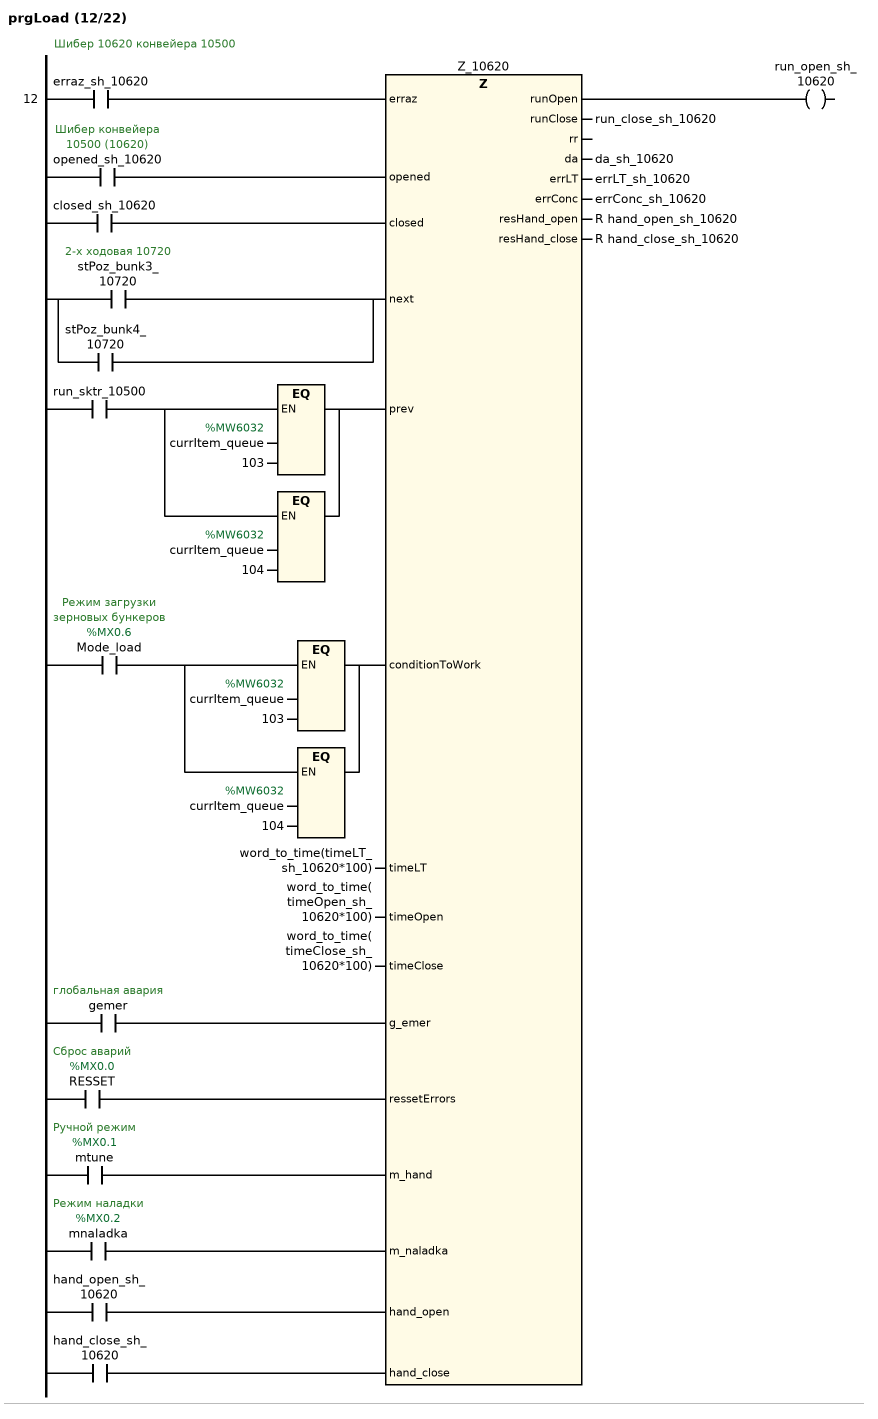
// NETWORK 12
// Шибер 10620 конвейера 10500
//   opened_sh_10620: Шибер конвейера 10500 (10620)
//   stPoz_bunk3_10720: 2-х ходовая 10720
//   currItem_queue: Текущий бункер для загрузки в очереди | AT %MW6032
//   Mode_load: Режим загрузки зерновых бункеров | AT %MX0.6
//   gemer: глобальная авария
//   RESSET: Сброс аварий | AT %MX0.0
//   mtune: Ручной режим | AT %MX0.1
//   mnaladka: Режим наладки | AT %MX0.2
//   errLT_sh_10620: Шибер 10620
Z_10620(
    erraz := erraz_sh_10620,
    opened := opened_sh_10620,
    closed := closed_sh_10620,
    next := stPoz_bunk3_10720 OR stPoz_bunk4_10720,
    prev := run_sktr_10500 AND currItem_queue = 103 OR run_sktr_10500 AND currItem_queue = 104,
    conditionToWork := Mode_load AND currItem_queue = 103 OR Mode_load AND currItem_queue = 104,
    timeLT := word_to_time(timeLT_sh_10620*100),
    timeOpen := word_to_time(timeOpen_sh_10620*100),
    timeClose := word_to_time(timeClose_sh_10620*100),
    g_emer := gemer,
    ressetErrors := RESSET,
    m_hand := mtune,
    m_naladka := mnaladka,
    hand_open := hand_open_sh_10620,
    hand_close := hand_close_sh_10620,
    runClose => run_close_sh_10620,
    da => da_sh_10620,
    errLT => errLT_sh_10620,
    errConc => errConc_sh_10620); // Z
hand_open_sh_10620 R= Z_10620.resHand_open;
hand_close_sh_10620 R= Z_10620.resHand_close;
run_open_sh_10620 := Z_10620.runOpen;

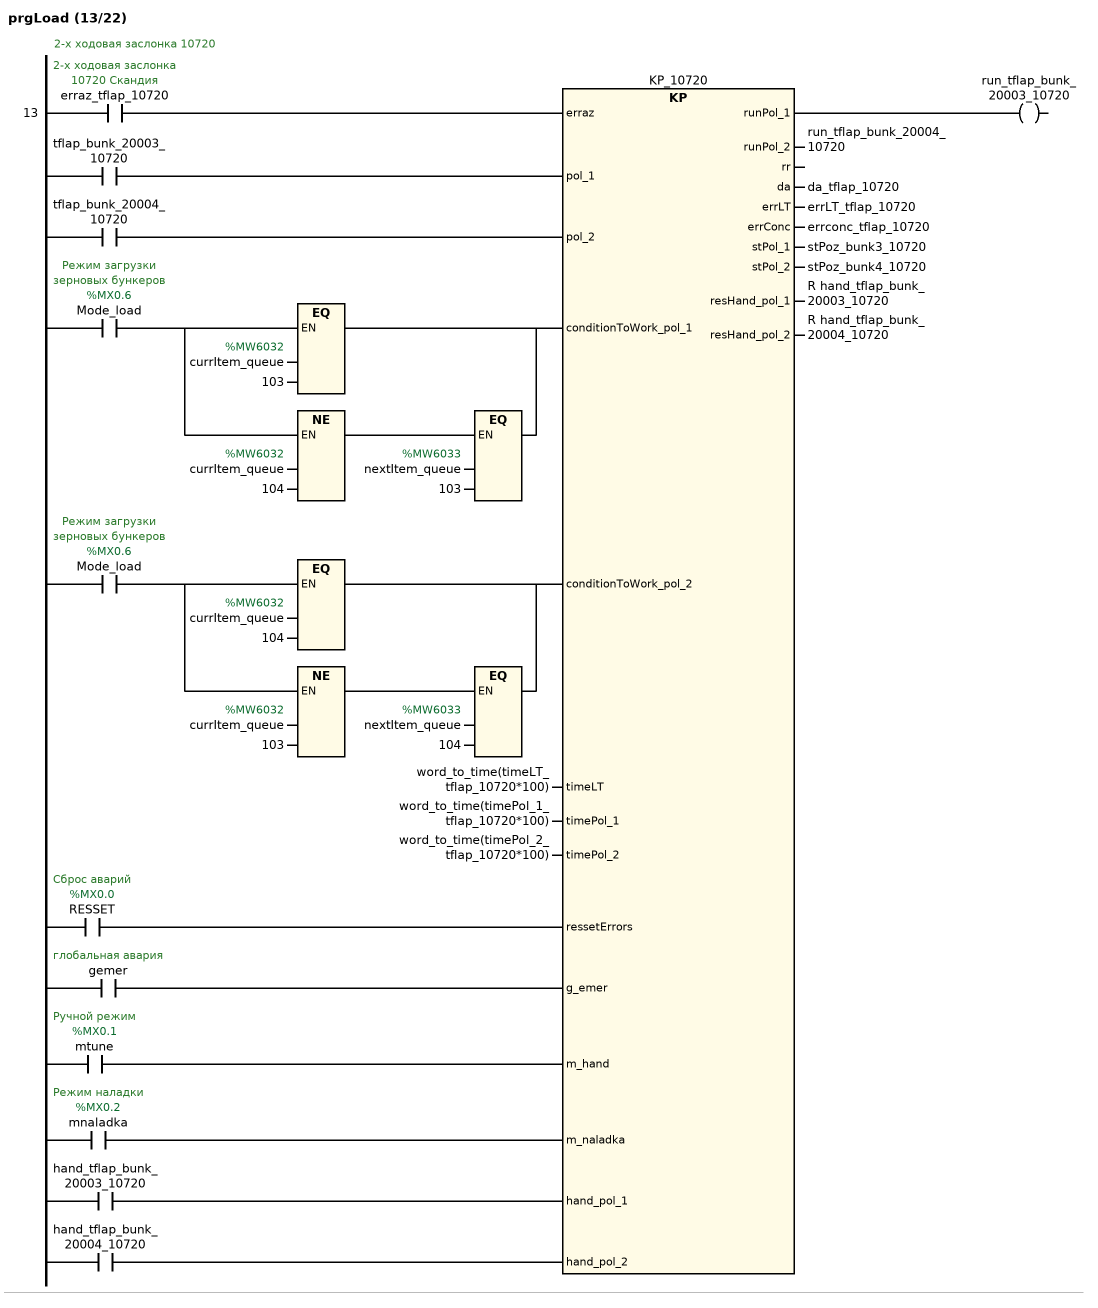
// NETWORK 13
// 2-х ходовая заслонка 10720
//   erraz_tflap_10720: 2-х ходовая заслонка 10720 Скандия
//   Mode_load: Режим загрузки зерновых бункеров | AT %MX0.6
//   currItem_queue: Текущий бункер для загрузки в очереди | AT %MW6032
//   nextItem_queue: Следующий бункер для загрузки в очереди | AT %MW6033
//   RESSET: Сброс аварий | AT %MX0.0
//   gemer: глобальная авария
//   mtune: Ручной режим | AT %MX0.1
//   mnaladka: Режим наладки | AT %MX0.2
//   errLT_tflap_10720: 2-х ходовой клапан КП_10720
//   stPoz_bunk3_10720: 2-х ходовая 10720
KP_10720(
    erraz := erraz_tflap_10720,
    pol_1 := tflap_bunk_20003_10720,
    pol_2 := tflap_bunk_20004_10720,
    conditionToWork_pol_1 := Mode_load AND currItem_queue = 103 OR Mode_load AND currItem_queue <> 104 AND nextItem_queue = 103,
    conditionToWork_pol_2 := Mode_load AND currItem_queue = 104 OR Mode_load AND currItem_queue <> 103 AND nextItem_queue = 104,
    timeLT := word_to_time(timeLT_tflap_10720*100),
    timePol_1 := word_to_time(timePol_1_tflap_10720*100),
    timePol_2 := word_to_time(timePol_2_tflap_10720*100),
    ressetErrors := RESSET,
    g_emer := gemer,
    m_hand := mtune,
    m_naladka := mnaladka,
    hand_pol_1 := hand_tflap_bunk_20003_10720,
    hand_pol_2 := hand_tflap_bunk_20004_10720,
    runPol_2 => run_tflap_bunk_20004_10720,
    da => da_tflap_10720,
    errLT => errLT_tflap_10720,
    errConc => errconc_tflap_10720,
    stPol_1 => stPoz_bunk3_10720,
    stPol_2 => stPoz_bunk4_10720); // KP
hand_tflap_bunk_20003_10720 R= KP_10720.resHand_pol_1;
hand_tflap_bunk_20004_10720 R= KP_10720.resHand_pol_2;
run_tflap_bunk_20003_10720 := KP_10720.runPol_1;

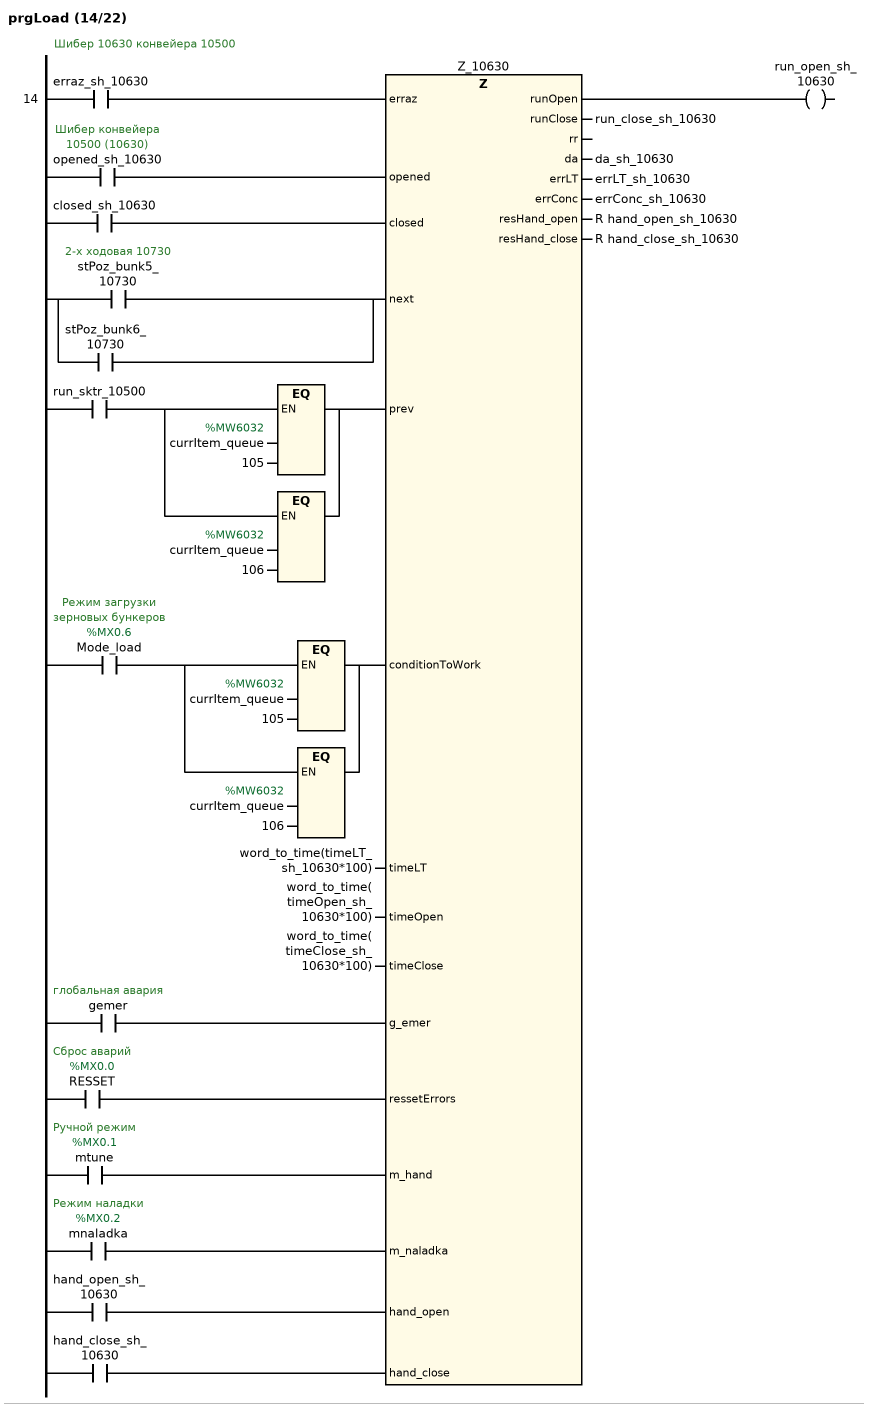
// NETWORK 14
// Шибер 10630 конвейера 10500
//   opened_sh_10630: Шибер конвейера 10500 (10630)
//   stPoz_bunk5_10730: 2-х ходовая 10730
//   currItem_queue: Текущий бункер для загрузки в очереди | AT %MW6032
//   Mode_load: Режим загрузки зерновых бункеров | AT %MX0.6
//   gemer: глобальная авария
//   RESSET: Сброс аварий | AT %MX0.0
//   mtune: Ручной режим | AT %MX0.1
//   mnaladka: Режим наладки | AT %MX0.2
//   errLT_sh_10630: Шибер 10630
Z_10630(
    erraz := erraz_sh_10630,
    opened := opened_sh_10630,
    closed := closed_sh_10630,
    next := stPoz_bunk5_10730 OR stPoz_bunk6_10730,
    prev := run_sktr_10500 AND currItem_queue = 105 OR run_sktr_10500 AND currItem_queue = 106,
    conditionToWork := Mode_load AND currItem_queue = 105 OR Mode_load AND currItem_queue = 106,
    timeLT := word_to_time(timeLT_sh_10630*100),
    timeOpen := word_to_time(timeOpen_sh_10630*100),
    timeClose := word_to_time(timeClose_sh_10630*100),
    g_emer := gemer,
    ressetErrors := RESSET,
    m_hand := mtune,
    m_naladka := mnaladka,
    hand_open := hand_open_sh_10630,
    hand_close := hand_close_sh_10630,
    runClose => run_close_sh_10630,
    da => da_sh_10630,
    errLT => errLT_sh_10630,
    errConc => errConc_sh_10630); // Z
hand_open_sh_10630 R= Z_10630.resHand_open;
hand_close_sh_10630 R= Z_10630.resHand_close;
run_open_sh_10630 := Z_10630.runOpen;

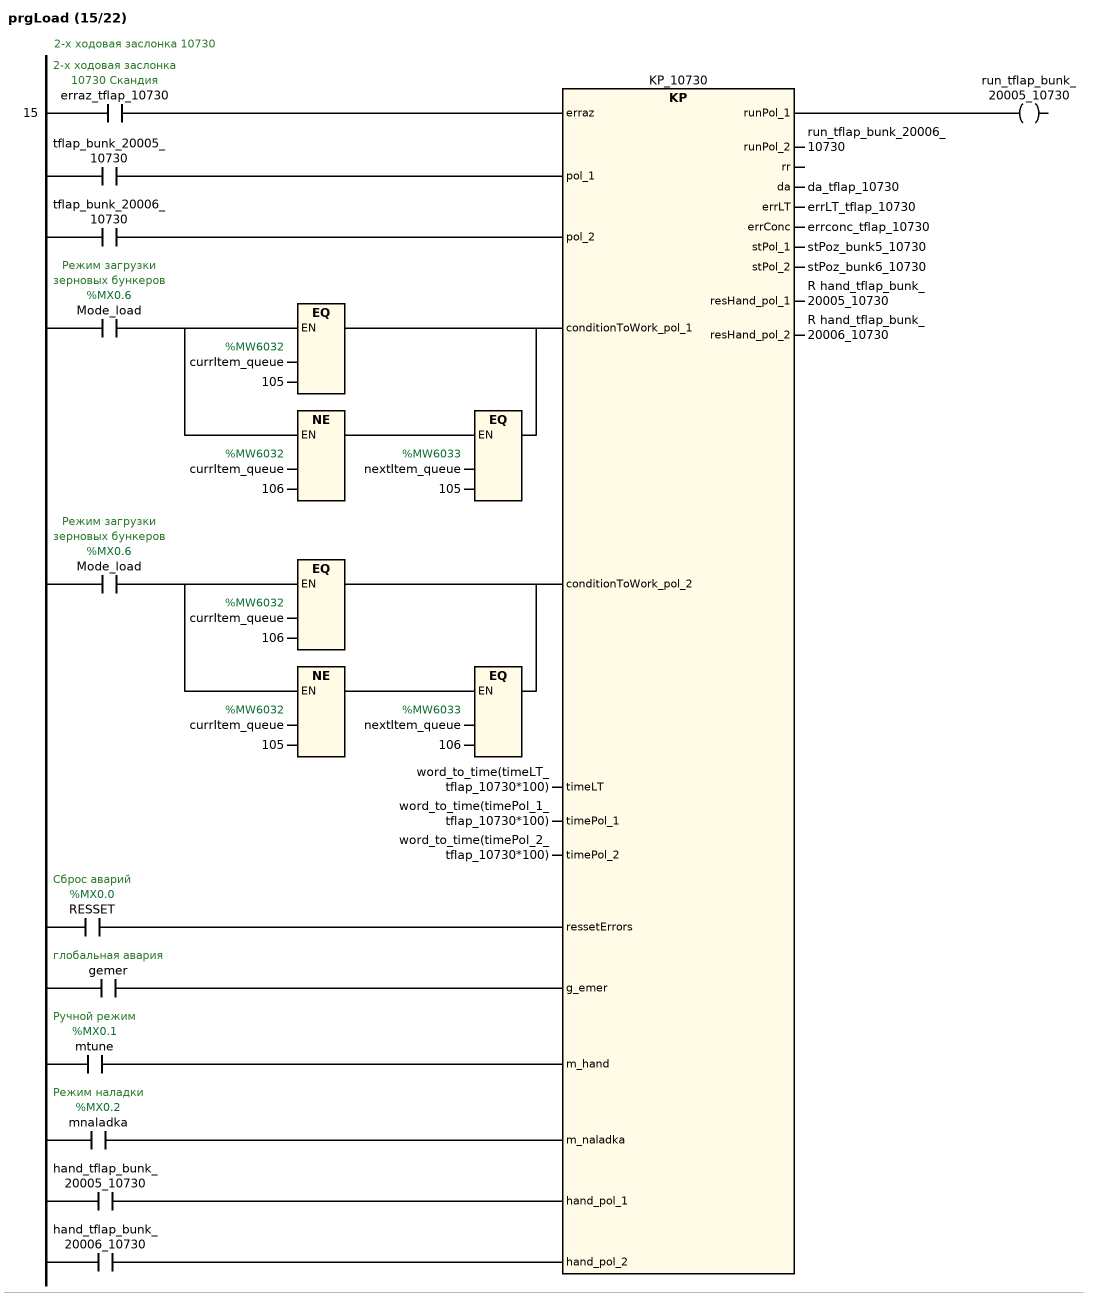
// NETWORK 15
// 2-х ходовая заслонка 10730
//   erraz_tflap_10730: 2-х ходовая заслонка 10730 Скандия
//   Mode_load: Режим загрузки зерновых бункеров | AT %MX0.6
//   currItem_queue: Текущий бункер для загрузки в очереди | AT %MW6032
//   nextItem_queue: Следующий бункер для загрузки в очереди | AT %MW6033
//   RESSET: Сброс аварий | AT %MX0.0
//   gemer: глобальная авария
//   mtune: Ручной режим | AT %MX0.1
//   mnaladka: Режим наладки | AT %MX0.2
//   errLT_tflap_10730: 2-х ходовой клапан КП_10730
//   stPoz_bunk5_10730: 2-х ходовая 10730
KP_10730(
    erraz := erraz_tflap_10730,
    pol_1 := tflap_bunk_20005_10730,
    pol_2 := tflap_bunk_20006_10730,
    conditionToWork_pol_1 := Mode_load AND currItem_queue = 105 OR Mode_load AND currItem_queue <> 106 AND nextItem_queue = 105,
    conditionToWork_pol_2 := Mode_load AND currItem_queue = 106 OR Mode_load AND currItem_queue <> 105 AND nextItem_queue = 106,
    timeLT := word_to_time(timeLT_tflap_10730*100),
    timePol_1 := word_to_time(timePol_1_tflap_10730*100),
    timePol_2 := word_to_time(timePol_2_tflap_10730*100),
    ressetErrors := RESSET,
    g_emer := gemer,
    m_hand := mtune,
    m_naladka := mnaladka,
    hand_pol_1 := hand_tflap_bunk_20005_10730,
    hand_pol_2 := hand_tflap_bunk_20006_10730,
    runPol_2 => run_tflap_bunk_20006_10730,
    da => da_tflap_10730,
    errLT => errLT_tflap_10730,
    errConc => errconc_tflap_10730,
    stPol_1 => stPoz_bunk5_10730,
    stPol_2 => stPoz_bunk6_10730); // KP
hand_tflap_bunk_20005_10730 R= KP_10730.resHand_pol_1;
hand_tflap_bunk_20006_10730 R= KP_10730.resHand_pol_2;
run_tflap_bunk_20005_10730 := KP_10730.runPol_1;

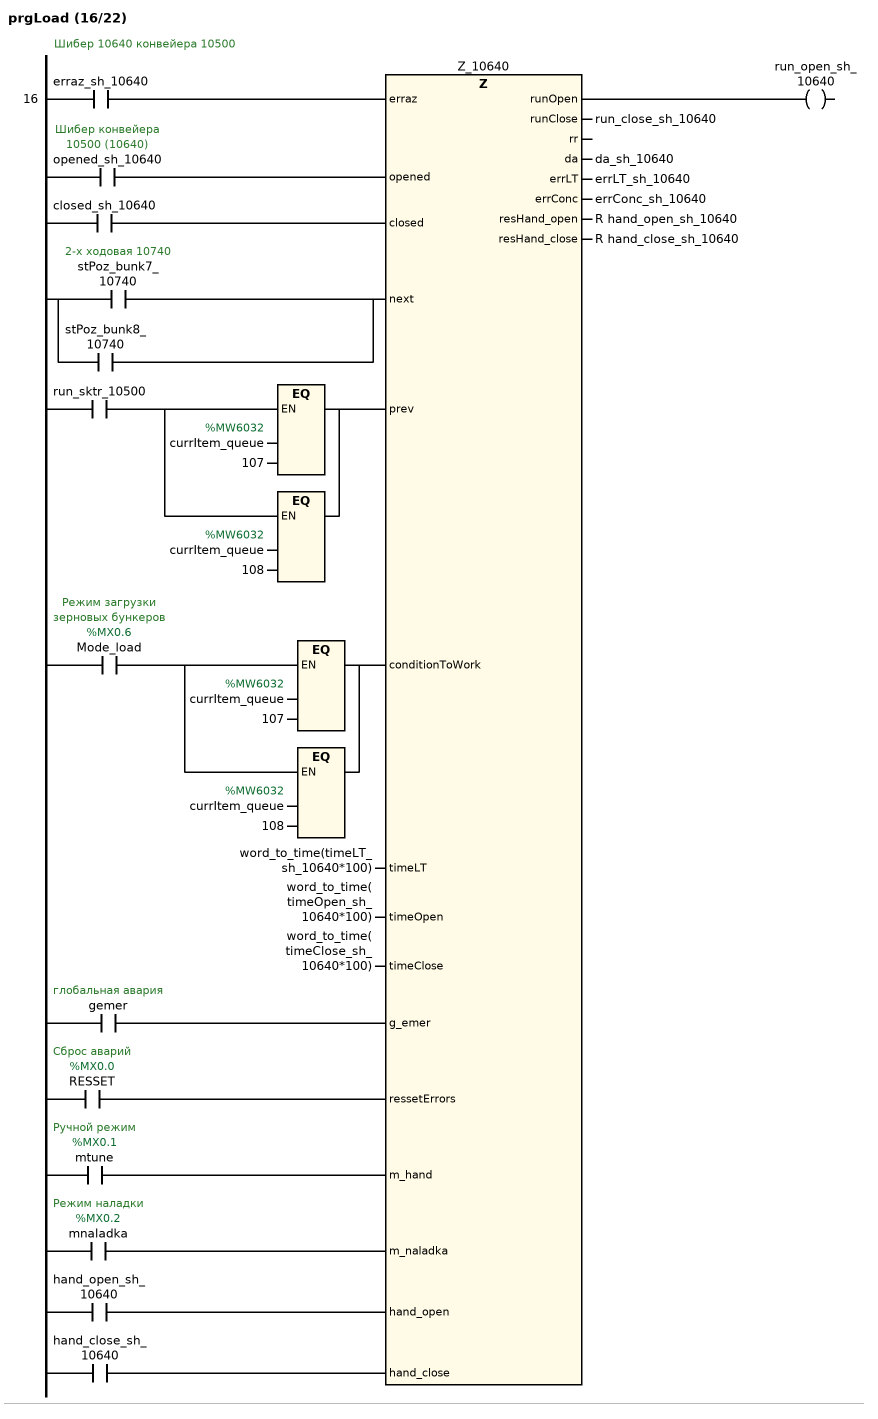
// NETWORK 16
// Шибер 10640 конвейера 10500
//   opened_sh_10640: Шибер конвейера 10500 (10640)
//   stPoz_bunk7_10740: 2-х ходовая 10740
//   currItem_queue: Текущий бункер для загрузки в очереди | AT %MW6032
//   Mode_load: Режим загрузки зерновых бункеров | AT %MX0.6
//   gemer: глобальная авария
//   RESSET: Сброс аварий | AT %MX0.0
//   mtune: Ручной режим | AT %MX0.1
//   mnaladka: Режим наладки | AT %MX0.2
//   errLT_sh_10640: Шибер 10640
Z_10640(
    erraz := erraz_sh_10640,
    opened := opened_sh_10640,
    closed := closed_sh_10640,
    next := stPoz_bunk7_10740 OR stPoz_bunk8_10740,
    prev := run_sktr_10500 AND currItem_queue = 107 OR run_sktr_10500 AND currItem_queue = 108,
    conditionToWork := Mode_load AND currItem_queue = 107 OR Mode_load AND currItem_queue = 108,
    timeLT := word_to_time(timeLT_sh_10640*100),
    timeOpen := word_to_time(timeOpen_sh_10640*100),
    timeClose := word_to_time(timeClose_sh_10640*100),
    g_emer := gemer,
    ressetErrors := RESSET,
    m_hand := mtune,
    m_naladka := mnaladka,
    hand_open := hand_open_sh_10640,
    hand_close := hand_close_sh_10640,
    runClose => run_close_sh_10640,
    da => da_sh_10640,
    errLT => errLT_sh_10640,
    errConc => errConc_sh_10640); // Z
hand_open_sh_10640 R= Z_10640.resHand_open;
hand_close_sh_10640 R= Z_10640.resHand_close;
run_open_sh_10640 := Z_10640.runOpen;

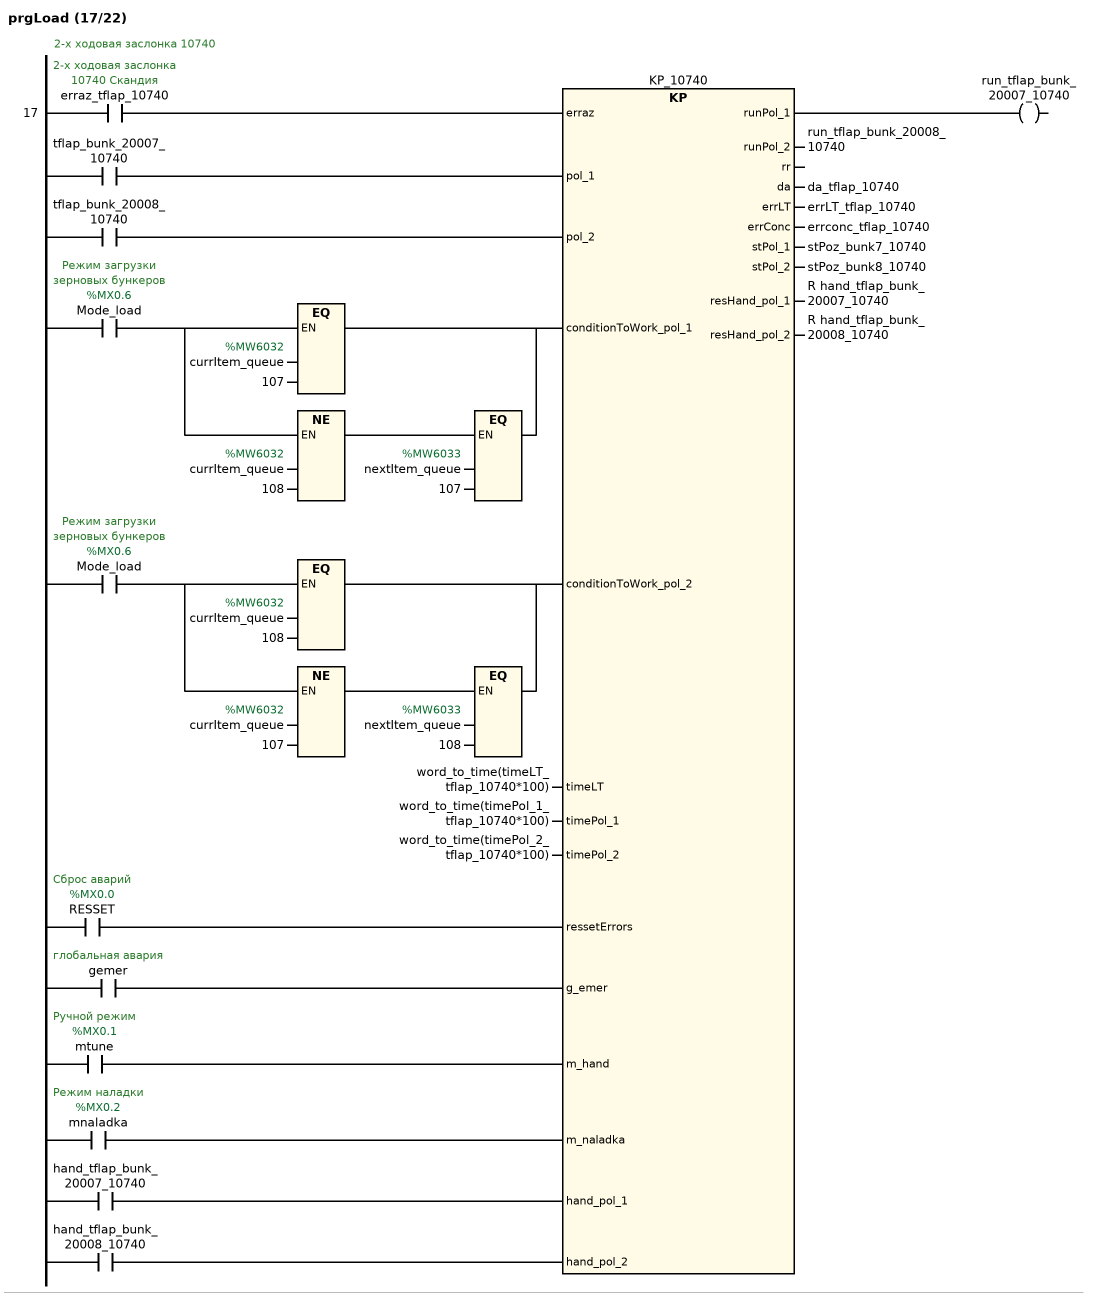
// NETWORK 17
// 2-х ходовая заслонка 10740
//   erraz_tflap_10740: 2-х ходовая заслонка 10740 Скандия
//   Mode_load: Режим загрузки зерновых бункеров | AT %MX0.6
//   currItem_queue: Текущий бункер для загрузки в очереди | AT %MW6032
//   nextItem_queue: Следующий бункер для загрузки в очереди | AT %MW6033
//   RESSET: Сброс аварий | AT %MX0.0
//   gemer: глобальная авария
//   mtune: Ручной режим | AT %MX0.1
//   mnaladka: Режим наладки | AT %MX0.2
//   errLT_tflap_10740: 2-х ходовой клапан КП_10740
//   stPoz_bunk7_10740: 2-х ходовая 10740
KP_10740(
    erraz := erraz_tflap_10740,
    pol_1 := tflap_bunk_20007_10740,
    pol_2 := tflap_bunk_20008_10740,
    conditionToWork_pol_1 := Mode_load AND currItem_queue = 107 OR Mode_load AND currItem_queue <> 108 AND nextItem_queue = 107,
    conditionToWork_pol_2 := Mode_load AND currItem_queue = 108 OR Mode_load AND currItem_queue <> 107 AND nextItem_queue = 108,
    timeLT := word_to_time(timeLT_tflap_10740*100),
    timePol_1 := word_to_time(timePol_1_tflap_10740*100),
    timePol_2 := word_to_time(timePol_2_tflap_10740*100),
    ressetErrors := RESSET,
    g_emer := gemer,
    m_hand := mtune,
    m_naladka := mnaladka,
    hand_pol_1 := hand_tflap_bunk_20007_10740,
    hand_pol_2 := hand_tflap_bunk_20008_10740,
    runPol_2 => run_tflap_bunk_20008_10740,
    da => da_tflap_10740,
    errLT => errLT_tflap_10740,
    errConc => errconc_tflap_10740,
    stPol_1 => stPoz_bunk7_10740,
    stPol_2 => stPoz_bunk8_10740); // KP
hand_tflap_bunk_20007_10740 R= KP_10740.resHand_pol_1;
hand_tflap_bunk_20008_10740 R= KP_10740.resHand_pol_2;
run_tflap_bunk_20007_10740 := KP_10740.runPol_1;

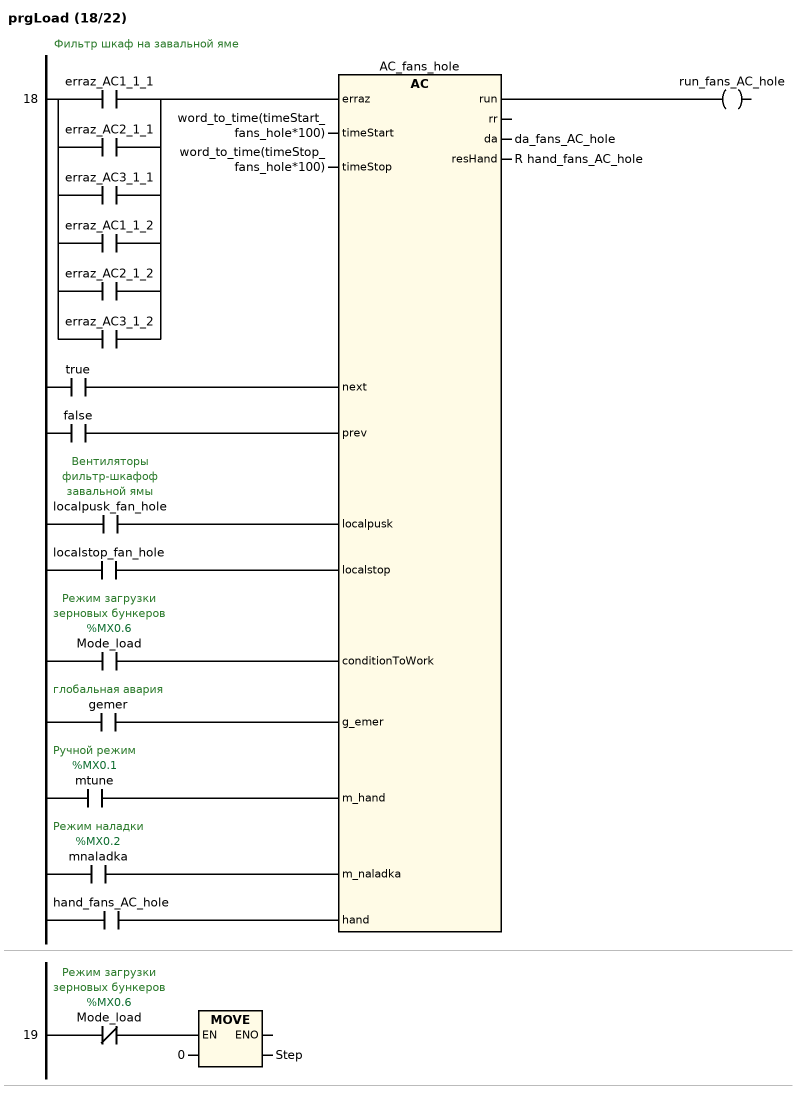
// NETWORK 18
// Фильтр шкаф на завальной яме
//   localpusk_fan_hole: Вентиляторы фильтр-шкафоф завальной ямы
//   Mode_load: Режим загрузки зерновых бункеров | AT %MX0.6
//   gemer: глобальная авария
//   mtune: Ручной режим | AT %MX0.1
//   mnaladka: Режим наладки | AT %MX0.2
AC_fans_hole(
    erraz := erraz_AC1_1_1 OR erraz_AC2_1_1 OR erraz_AC3_1_1 OR erraz_AC1_1_2 OR erraz_AC2_1_2 OR erraz_AC3_1_2,
    timeStart := word_to_time(timeStart_fans_hole*100),
    timeStop := word_to_time(timeStop_fans_hole*100),
    next := true,
    prev := false,
    localpusk := localpusk_fan_hole,
    localstop := localstop_fan_hole,
    conditionToWork := Mode_load,
    g_emer := gemer,
    m_hand := mtune,
    m_naladka := mnaladka,
    hand := hand_fans_AC_hole,
    da => da_fans_AC_hole); // AC
hand_fans_AC_hole R= AC_fans_hole.resHand;
run_fans_AC_hole := AC_fans_hole.run;

// NETWORK 19
//   Mode_load: Режим загрузки зерновых бункеров | AT %MX0.6
IF NOT Mode_load THEN Step := 0; END_IF

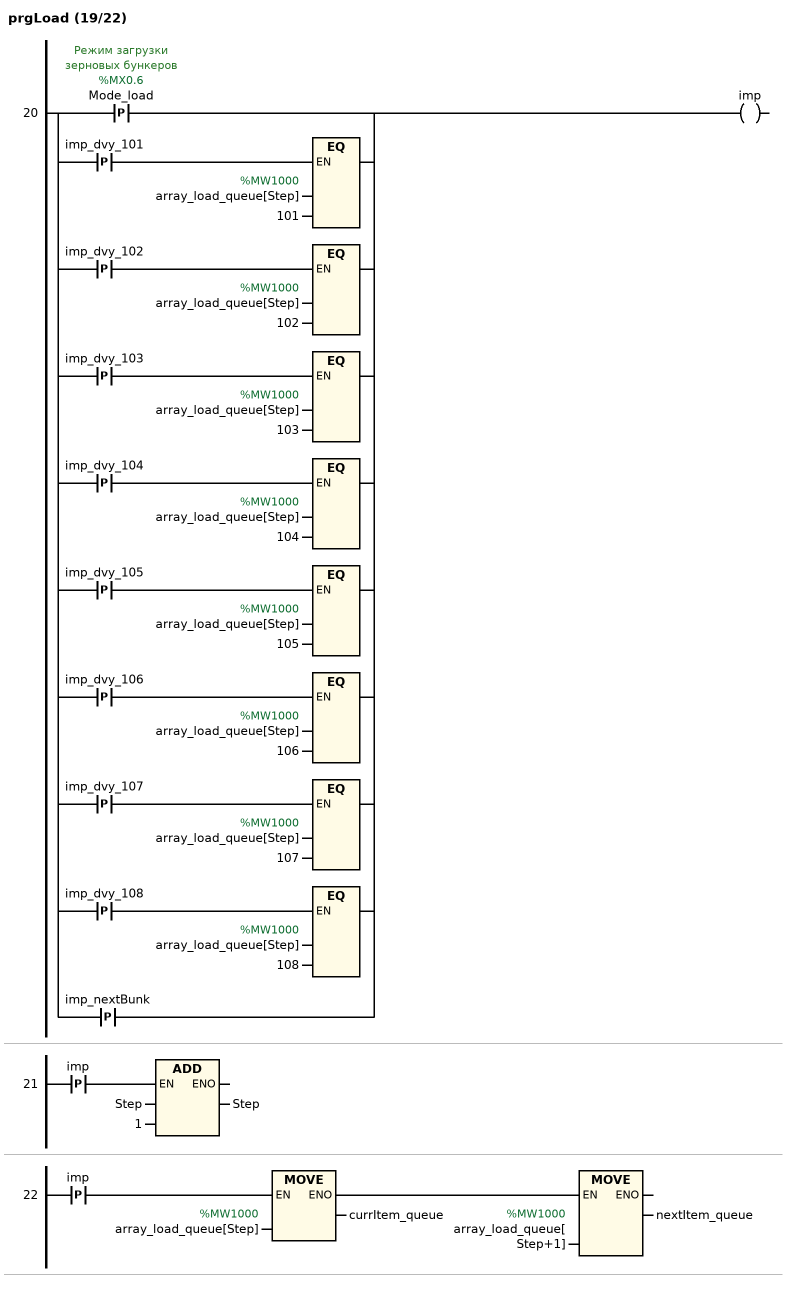
// NETWORK 20
//   Mode_load: Режим загрузки зерновых бункеров | AT %MX0.6
//   array_load_queue[Step]: Массив очереди загрузки зерновых бункеров | AT %MW1000
_rt1(CLK := Mode_load);
_rt2(CLK := imp_dvy_101);
_rt3(CLK := imp_dvy_102);
_rt4(CLK := imp_dvy_103);
_rt5(CLK := imp_dvy_104);
_rt6(CLK := imp_dvy_105);
_rt7(CLK := imp_dvy_106);
_rt8(CLK := imp_dvy_107);
_rt9(CLK := imp_dvy_108);
_rt10(CLK := imp_nextBunk);
imp := _rt1.Q OR _rt2.Q AND array_load_queue[Step] = 101 OR _rt3.Q AND array_load_queue[Step] = 102 OR _rt4.Q AND array_load_queue[Step] = 103 OR _rt5.Q AND array_load_queue[Step] = 104 OR _rt6.Q AND array_load_queue[Step] = 105 OR _rt7.Q AND array_load_queue[Step] = 106 OR _rt8.Q AND array_load_queue[Step] = 107 OR _rt9.Q AND array_load_queue[Step] = 108 OR _rt10.Q;

// NETWORK 21
_rt11(CLK := imp);
IF _rt11.Q THEN Step := Step + 1; END_IF

// NETWORK 22
//   array_load_queue[Step]: Массив очереди загрузки зерновых бункеров | AT %MW1000
//   currItem_queue: Текущий бункер для загрузки в очереди | AT %MW6032
//   array_load_queue[Step+1]: Массив очереди загрузки зерновых бункеров | AT %MW1000
//   nextItem_queue: Следующий бункер для загрузки в очереди | AT %MW6033
_rt12(CLK := imp);
_w1 := _rt12.Q;
IF _w1 THEN currItem_queue := array_load_queue[Step]; END_IF
IF _w1 THEN nextItem_queue := array_load_queue[Step+1]; END_IF

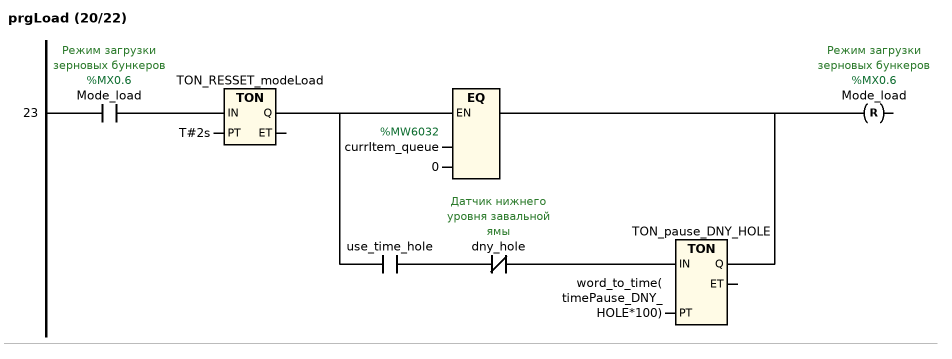
// NETWORK 23
//   Mode_load: Режим загрузки зерновых бункеров | AT %MX0.6
//   currItem_queue: Текущий бункер для загрузки в очереди | AT %MW6032
//   dny_hole: Датчик нижнего уровня завальной ямы
TON_RESSET_modeLoad(IN := Mode_load, PT := T#2s); // TON
TON_pause_DNY_HOLE(IN := (TON_RESSET_modeLoad.Q AND use_time_hole) AND NOT dny_hole, PT := word_to_time(timePause_DNY_HOLE*100)); // TON
Mode_load R= TON_RESSET_modeLoad.Q AND currItem_queue = 0 OR TON_pause_DNY_HOLE.Q;

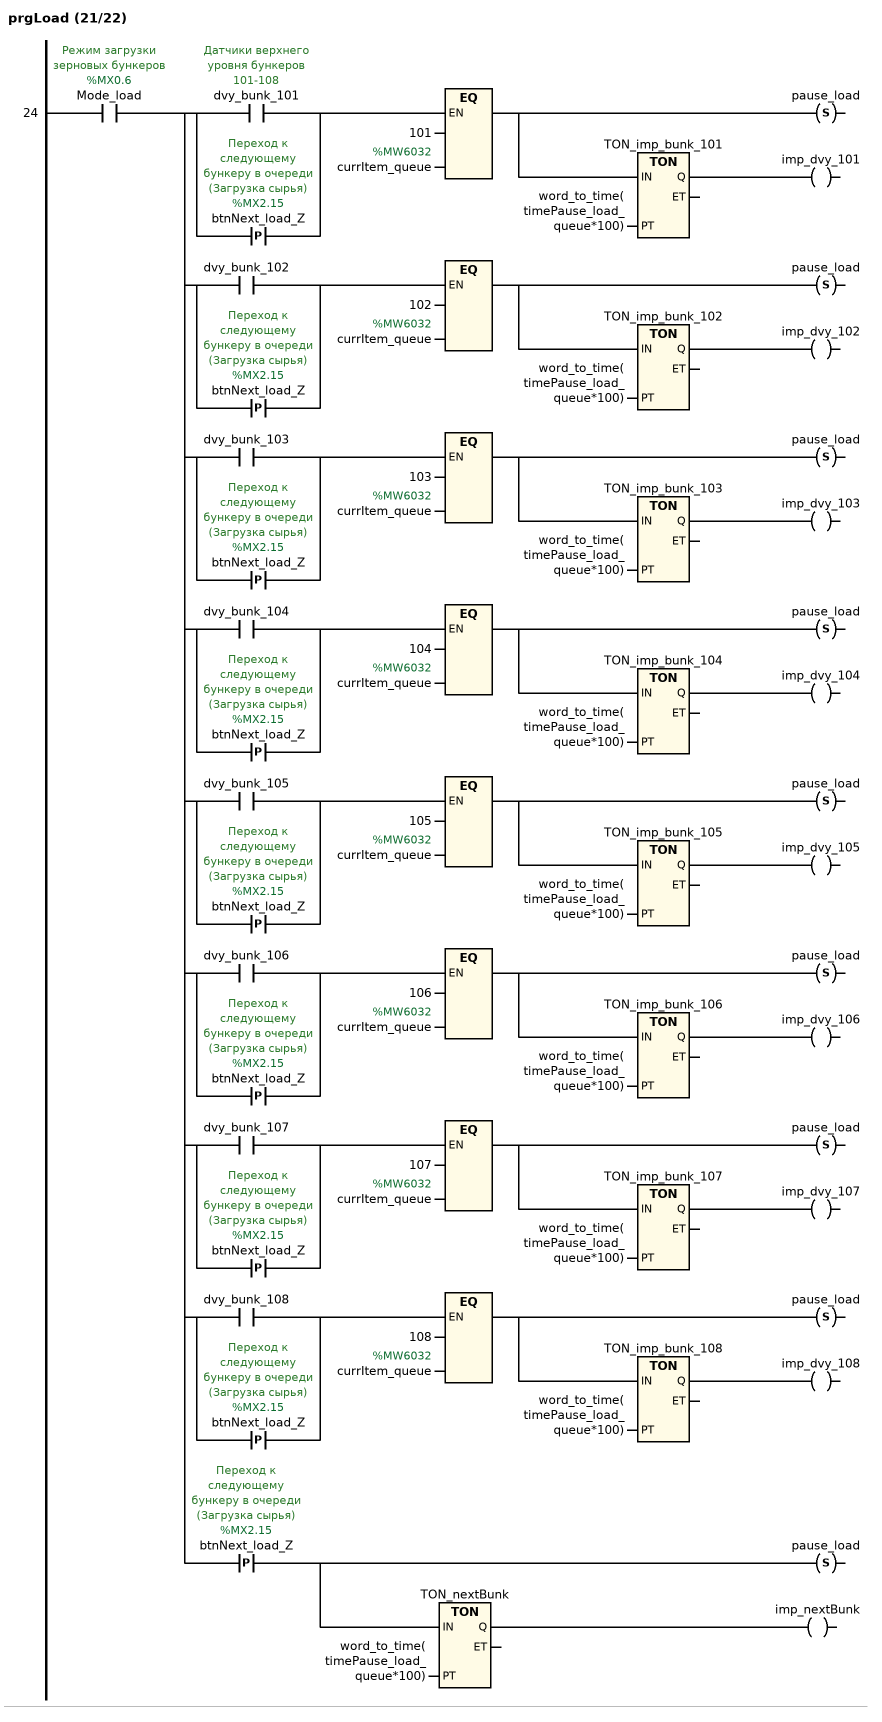
// NETWORK 24
//   Mode_load: Режим загрузки зерновых бункеров | AT %MX0.6
//   dvy_bunk_101: Датчики верхнего уровня бункеров 101-108
//   btnNext_load_Z: Переход к следующему бункеру в очереди (Загрузка сырья) | AT %MX2.15
//   currItem_queue: Текущий бункер для загрузки в очереди | AT %MW6032
_rt13(CLK := btnNext_load_Z);
_w2 := Mode_load AND (dvy_bunk_101 OR _rt13.Q) AND 101 = currItem_queue;
pause_load S= _w2;
TON_imp_bunk_101(IN := _w2, PT := word_to_time(timePause_load_queue*100)); // TON
imp_dvy_101 := TON_imp_bunk_101.Q;
_rt14(CLK := btnNext_load_Z);
_w3 := Mode_load AND (dvy_bunk_102 OR _rt14.Q) AND 102 = currItem_queue;
pause_load S= _w3;
TON_imp_bunk_102(IN := _w3, PT := word_to_time(timePause_load_queue*100)); // TON
imp_dvy_102 := TON_imp_bunk_102.Q;
_rt15(CLK := btnNext_load_Z);
_w4 := Mode_load AND (dvy_bunk_103 OR _rt15.Q) AND 103 = currItem_queue;
pause_load S= _w4;
TON_imp_bunk_103(IN := _w4, PT := word_to_time(timePause_load_queue*100)); // TON
imp_dvy_103 := TON_imp_bunk_103.Q;
_rt16(CLK := btnNext_load_Z);
_w5 := Mode_load AND (dvy_bunk_104 OR _rt16.Q) AND 104 = currItem_queue;
pause_load S= _w5;
TON_imp_bunk_104(IN := _w5, PT := word_to_time(timePause_load_queue*100)); // TON
imp_dvy_104 := TON_imp_bunk_104.Q;
_rt17(CLK := btnNext_load_Z);
_w6 := Mode_load AND (dvy_bunk_105 OR _rt17.Q) AND 105 = currItem_queue;
pause_load S= _w6;
TON_imp_bunk_105(IN := _w6, PT := word_to_time(timePause_load_queue*100)); // TON
imp_dvy_105 := TON_imp_bunk_105.Q;
_rt18(CLK := btnNext_load_Z);
_w7 := Mode_load AND (dvy_bunk_106 OR _rt18.Q) AND 106 = currItem_queue;
pause_load S= _w7;
TON_imp_bunk_106(IN := _w7, PT := word_to_time(timePause_load_queue*100)); // TON
imp_dvy_106 := TON_imp_bunk_106.Q;
_rt19(CLK := btnNext_load_Z);
_w8 := Mode_load AND (dvy_bunk_107 OR _rt19.Q) AND 107 = currItem_queue;
pause_load S= _w8;
TON_imp_bunk_107(IN := _w8, PT := word_to_time(timePause_load_queue*100)); // TON
imp_dvy_107 := TON_imp_bunk_107.Q;
_rt20(CLK := btnNext_load_Z);
_w9 := Mode_load AND (dvy_bunk_108 OR _rt20.Q) AND 108 = currItem_queue;
pause_load S= _w9;
TON_imp_bunk_108(IN := _w9, PT := word_to_time(timePause_load_queue*100)); // TON
imp_dvy_108 := TON_imp_bunk_108.Q;
_rt21(CLK := btnNext_load_Z);
_w10 := Mode_load AND _rt21.Q;
pause_load S= _w10;
TON_nextBunk(IN := _w10, PT := word_to_time(timePause_load_queue*100)); // TON
imp_nextBunk := TON_nextBunk.Q;

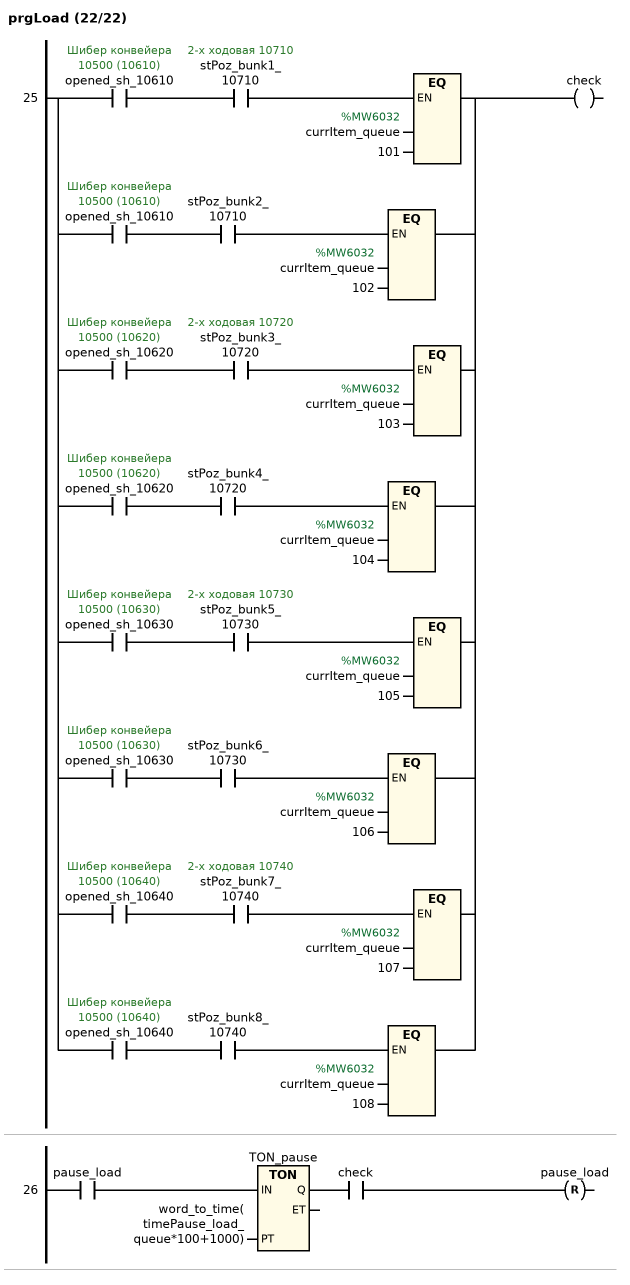
// NETWORK 25
//   opened_sh_10610: Шибер конвейера 10500 (10610)
//   stPoz_bunk1_10710: 2-х ходовая 10710
//   currItem_queue: Текущий бункер для загрузки в очереди | AT %MW6032
//   opened_sh_10620: Шибер конвейера 10500 (10620)
//   stPoz_bunk3_10720: 2-х ходовая 10720
//   opened_sh_10630: Шибер конвейера 10500 (10630)
//   stPoz_bunk5_10730: 2-х ходовая 10730
//   opened_sh_10640: Шибер конвейера 10500 (10640)
//   stPoz_bunk7_10740: 2-х ходовая 10740
check := opened_sh_10610 AND stPoz_bunk1_10710 AND currItem_queue = 101 OR (opened_sh_10610 AND stPoz_bunk2_10710 AND currItem_queue = 102 OR (opened_sh_10620 AND stPoz_bunk3_10720 AND currItem_queue = 103 OR (opened_sh_10620 AND stPoz_bunk4_10720 AND currItem_queue = 104 OR (opened_sh_10630 AND stPoz_bunk5_10730 AND currItem_queue = 105 OR opened_sh_10630 AND stPoz_bunk6_10730 AND currItem_queue = 106 OR opened_sh_10640 AND stPoz_bunk7_10740 AND currItem_queue = 107 OR opened_sh_10640 AND stPoz_bunk8_10740 AND currItem_queue = 108))));

// NETWORK 26
TON_pause(IN := pause_load, PT := word_to_time(timePause_load_queue*100+1000)); // TON
pause_load R= TON_pause.Q AND check;

END_PROGRAM

// PLC_241/Application/FB/SKTR/T
FUNCTION_BLOCK T
VAR_INPUT
	dks: BOOL;
	dp: BOOL;
	localpusk: BOOL;
	localstop: BOOL;
	erraz: BOOL;
	timeDKS: TIME;
	timeDP: TIME;
	next: BOOL;
	prev: BOOL;
	conditionToWork: BOOL;
	timeStart: TIME;
	timeStop: TIME;
	ressetErrors: BOOL;
	g_emer: BOOL;
	m_hand: BOOL;
	m_naladka: BOOL;
	hand: BOOL;
	offdks: BOOL;
	offdp: BOOL;
END_VAR
VAR_OUTPUT
	run: BOOL;
	rr: BOOL;
	da: BOOL;
	errDKS: BOOL;
	errDP: BOOL;
	resHand: BOOL;
END_VAR
VAR
	TON_DKS1: TON;
	TON_DKS2: TON;
	TON_DP: TON;
	TON_start: TON;
	start: BOOL;
	TON_stop: TON;
END_VAR
VAR // added by the converter: edge detectors and wires of the graphical bodies
    _w1 : BOOL;
END_VAR

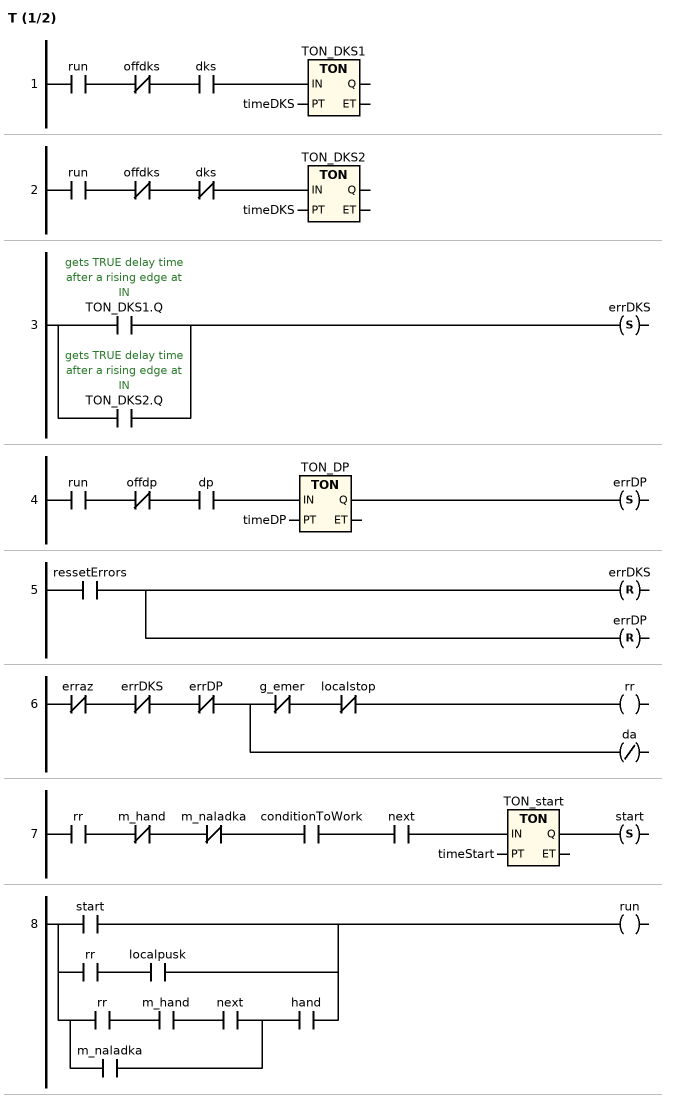
// NETWORK 1
TON_DKS1(IN := run AND NOT offdks AND dks, PT := timeDKS); // TON

// NETWORK 2
TON_DKS2(IN := run AND NOT offdks AND NOT dks, PT := timeDKS); // TON

// NETWORK 3
//   TON_DKS1.Q: gets TRUE delay time after a rising edge at IN
//   TON_DKS2.Q: gets TRUE delay time after a rising edge at IN
errDKS S= TON_DKS1.Q OR TON_DKS2.Q;

// NETWORK 4
TON_DP(IN := run AND NOT offdp AND dp, PT := timeDP); // TON
errDP S= TON_DP.Q;

// NETWORK 5
errDKS R= ressetErrors;
errDP R= ressetErrors;

// NETWORK 6
_w1 := NOT erraz AND NOT errDKS AND NOT errDP;
rr := _w1 AND NOT g_emer AND NOT localstop;
da := NOT _w1;

// NETWORK 7
TON_start(IN := rr AND NOT m_hand AND NOT m_naladka AND conditionToWork AND next, PT := timeStart); // TON
start S= TON_start.Q;

// NETWORK 8
run := start OR rr AND localpusk OR (rr AND m_hand AND next OR m_naladka) AND hand;

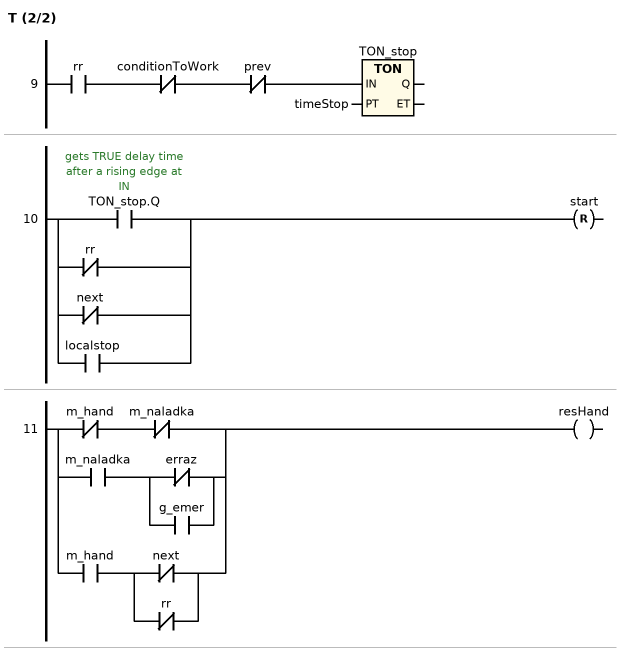
// NETWORK 9
TON_stop(IN := rr AND NOT conditionToWork AND NOT prev, PT := timeStop); // TON

// NETWORK 10
//   TON_stop.Q: gets TRUE delay time after a rising edge at IN
start R= TON_stop.Q OR NOT rr OR NOT next OR localstop;

// NETWORK 11
resHand := NOT m_hand AND NOT m_naladka OR m_naladka AND (NOT erraz OR g_emer) OR m_hand AND (NOT next OR NOT rr);

END_FUNCTION_BLOCK

// PLC_241/Application/FB/ASP/AC
FUNCTION_BLOCK AC
VAR_INPUT
	erraz: BOOL;
	timeStart: TIME;
	timeStop: TIME;
	next: BOOL;
	prev: BOOL;
	localpusk: BOOL;
	localstop: BOOL;
	conditionToWork: BOOL; 
	g_emer: BOOL;
	m_hand: BOOL;
	m_naladka: BOOL;
	hand: BOOL;
END_VAR
VAR_OUTPUT
	run: BOOL;
	rr: BOOL;
	da: BOOL;
	resHand: BOOL;
END_VAR
VAR
	TON_start: TON;
	start: BOOL;
	TON_0stop: TON;
	TON_stop: TON;
END_VAR
VAR // added by the converter: edge detectors and wires of the graphical bodies
    _w1 : BOOL;
END_VAR

